# B&R Automation Studio project Panasonic_LinkaPowerCP2_A2021055 (part 32)

#### Main.st - Init, cyclic, exit code
```iecst
PROGRAM _INIT

	//Init parametre serva zdvihu aplikatora//
	P4_Etiketovacka.ServoZdvihuAplikatora.Parameters.Override:= 100;
	P4_Etiketovacka.PAR.ZdvihAplikatora_JoggRychlost:= 5;
	P4_Etiketovacka.ServoZdvihuAplikatora.Command.TorqueLimitation:= TRUE;
	P4_Etiketovacka.ServoZdvihuAplikatora.Parameters.Torque:= 1.0;

END_PROGRAM

PROGRAM _CYCLIC

	//Volanie funkcie SequenceControl//
	SequenceControl(SC:= SC_P4_Etiketovacka);

	//Volanie podprogramov//
	OvlCentrovacky;
	OvlOtacaniaAplikatora;
	IOLinkKomunikacia;
	COM_Tlaciaren;
	VytvorenieEtikety;

	//Enable serva//
	IF Safety.STAV.P4_ZonaBunky_AKTIVNA AND NOT P4_Etiketovacka.ServoZdvihuAplikatora.Command.ErrReset THEN
		P4_Etiketovacka.ServoZdvihuAplikatora.Command.PowerON:= TRUE;
	ELSE
		P4_Etiketovacka.ServoZdvihuAplikatora.Command.PowerON:= FALSE;
	END_IF

	//Zaokrúhlenie aktuálnej pozície serva zdvihu//
	ServoZdvihu_AktualPosition_UDINT:= REAL_TO_UDINT(P4_Etiketovacka.ServoZdvihuAplikatora.Status.ActPosition);

	//Reset poruchy serva//
	IF EDGEPOS(Safety.STAV.P4_ZonaBunky_AKTIVNA)THEN
		P4_Etiketovacka.ServoZdvihuAplikatora.Command.ErrReset:= TRUE;
	END_IF

	CasResetServo_1.IN:= P4_Etiketovacka.ServoZdvihuAplikatora.Command.ErrReset;
	IF CasResetServo_1.Q AND NOT P4_Etiketovacka.ServoZdvihuAplikatora.Status.Error THEN
		P4_Etiketovacka.ServoZdvihuAplikatora.Command.ErrReset:= FALSE;
	END_IF

	CasResetServo_1.PT:= T#500ms;
	CasResetServo_1();

	//Reset sekcie //
	IF P4_Etiketovacka.Reset THEN
		SC_P4_Etiketovacka.Step:= 0;
		P4_Etiketovacka.ServoZdvihuAplikatora.Command.ErrReset:= TRUE;
		P4_Etiketovacka.Reset:= FALSE;
	ELSIF NOT Safety.STAV.Linka_ZonaCS_AKTIVNA AND NOT P4_Etiketovacka.Automat THEN
		SC_P4_Etiketovacka.Step:= 0;
	ELSIF NOT Safety.STAV.Linka_ZonaCS_AKTIVNA AND P4_Etiketovacka.Automat THEN
		P4_Pracovisko.STAV.Porucha_ST5:= TRUE;
	END_IF

	//Ukončenie komunikácie pri poruche//
	IF P4_Pracovisko.STAV.Porucha_ST5 AND NOT Triger_0 THEN
		Triger_0:= TRUE;
		IF P4_Etiketovacka.STAV.VyrobaZacala THEN
			Paletka[i].PAR.StavPowerCP:= 'FAIL';
			Paletka[i].STAV.StavPaletky:= 'NG';
			P4_Etiketovacka.KoniecCyklu:= TRUE;
			SC_P4_Etiketovacka.ResetStep:= TRUE;
			SC_P4_Etiketovacka.Step:= 550;
		ELSE
			SC_P4_Etiketovacka.ResetStep:= TRUE;
			SC_P4_Etiketovacka.Step:= 0;
		END_IF
	END_IF

	IF NOT P4_Pracovisko.STAV.Porucha_ST5 THEN
		Triger_0:= FALSE;
	END_IF

	CASE SC_P4_Etiketovacka.Step OF

		0:
			SC_P4_Etiketovacka.StepName:='0 - Nulovanie';
			SC_OvlCentrovacky.Step:= 0;
			SC_OvlOtacaniaAplikatora.Step:= 0;
			P4_Etiketovacka.Automat:= FALSE;
			P4_Etiketovacka.KoniecCyklu:= FALSE;
			P4_Etiketovacka.Manual:= FALSE;
			P4_Etiketovacka.STAV.PoINIT:= FALSE;
			P4_Etiketovacka.STAV.VyrobaZacala:= FALSE;
			P4_Etiketovacka.STAV.VstupnaKamerovaKontrola:= FALSE;
			P4_Etiketovacka.OUT.ZasunStoper:= FALSE;
			P4_Etiketovacka.OUT.Centrovanie_VYSUN:= FALSE;
			P4_Etiketovacka.OUT.Centrovanie_ZASUN:= TRUE;
			P4_Etiketovacka.OUT.Aplikator_VYSUN:= FALSE;
			P4_Etiketovacka.OUT.Aplikator_OtocVPRED:= FALSE;
			P4_Etiketovacka.OUT.Aplikator_OtocVZAD:= FALSE;
			P4_Etiketovacka.OUT.OfukEtikety_ON:= FALSE;
			P4_Etiketovacka.OUT.PritlakPowerCP_VYSUN:= FALSE;
			P4_Etiketovacka.OUT.PrisavanieEtikety_ON:= FALSE;
			P4_Etiketovacka.OUT.PrisavanieEtikety_OFF:= TRUE;
			P4_Etiketovacka.RFID_hlava.PrecitajChipRFID:= FALSE;

			P4_Etiketovacka.ServoZdvihuAplikatora.Command.JogNeg:= FALSE;
			P4_Etiketovacka.ServoZdvihuAplikatora.Command.JogPos:= FALSE;
			P4_Etiketovacka.ServoZdvihuAplikatora.Command.MoveAdditive:= FALSE;
			P4_Etiketovacka.ServoZdvihuAplikatora.Command.MovePosition:= FALSE;
			IF NOT P4_Etiketovacka.ServoZdvihuAplikatora.Status.StandStill THEN
				P4_Etiketovacka.ServoZdvihuAplikatora.Command.Stop:= TRUE;
			END_IF

			P4_Etiketovacka.CMD.RR_ZdvihAplikatora_DOLE:= FALSE;
			P4_Etiketovacka.CMD.RR_ZdvihAplikatora_HORE:= FALSE;
			P4_Etiketovacka.CMD.RR_NalepEtiketu:= FALSE;
			P4_Etiketovacka.STAV.RR_SekvenciaEtiketovania_BUSY:= FALSE;
			P4_Etiketovacka.CMD.RR_VysunCentrovanie:= FALSE;
			P4_Etiketovacka.CMD.RR_PrisavanieEtikety:= FALSE;

			CAM14.CMD.Triger:= FALSE;
			CAM14.STAV.Results_READY:= FALSE;

			CAM15.CMD.Triger:= FALSE;
			CAM15.STAV.Results_READY:= FALSE;
			FTP_CAM15.CMD.OdosliFotku:= FALSE;
			FTP_CAM15.CMD.VymazFotku:= FALSE;

			TRCB_P4_Etiketovacka_ST9.CMD.VyziadajStavPaletky_TYP1:= FALSE;
			TRCB_P4_Etiketovacka_ST9.CMD.PriradQRkodFiltra_TYP3:= FALSE;
			TRCB_P4_Etiketovacka_ST9.CMD.OdosliStavPaletky_TYP2:= FALSE;
			TRCB_P4_Etiketovacka_ST9.CMD.VyziadajCisloEtikety_TYP0:= FALSE;
			TRCB_P4_Etiketovacka_ST9.CMD.VyziadajStavPanatrace_TYP4:= FALSE;

			P4_Etiketov_KAM_Result_Ignoruj:= FALSE;
			P4_Etiketov_KAM_Result_OK:= FALSE;
			P4_Etiketov_KAM_Result_NG:= FALSE;
			P34_Vizu.ZobrazHL1_ST9:= FALSE;
			P34_Vizu.ZobrazHL2_ST9:= FALSE;
			P34_Vizu.ZobrazHL3_ST9:= FALSE;
			P34_Vizu.ZobrazHL4_ST9:= FALSE;
			TRCB_P4_Etiketov_OpatovnyDopyt:= FALSE;
			TRCB_P4_Etiketov_PaletkaNG:= FALSE;
			PocetTrigrovKamery:= 0;
			PocetDopytovNaServer:= 0;
			CisloFotky:= 0;
			TestovaciKus:= FALSE;
			P4_Etiketovacka.STAV.PowerCP_ZhodaQRkodu_OK:= FALSE;
			P4_Etiketovacka.STAV.Etiketa_ZhodaQRkodu_OK:= FALSE;
			P4_Etiketovacka.STAV.PrebiehaVyvezeniePaletky:= FALSE;
			P4_ZdvizkaZaFunkcTestA.STAV.PrebiehaVyvezeniePaletky:= FALSE;
			P4_Etiketovanie_Taktime.IN.START_MeraniaCasu:= FALSE;
			P4_Etiketovanie_Taktime.IN.START_MeraniaStratovehoCasu:= FALSE;

			Tlaciaren.CMD.VytlacEtiketu:= FALSE;

			IF Safety.STAV.Linka_ZonaCS_AKTIVNA AND
				Safety.STAV.P4_ZonaBunky_AKTIVNA AND
				(P4_Etiketovacka.ServoZdvihuAplikatora.Status.Ready AND P4_Etiketovacka.ServoZdvihuAplikatora.Status.StandStill) AND
				P4_Pracovisko.STAV.HardwareBunky_OK AND
				NOT P4_Pracovisko.STAV.Porucha_ST1 AND
				NOT P4_Pracovisko.STAV.Porucha_ST2 AND
				NOT P4_Pracovisko.STAV.Porucha_ST3 AND
				NOT P4_Pracovisko.STAV.Porucha_ST4 AND
				NOT P4_Pracovisko.STAV.Porucha_ST5 AND
				NOT P4_Pracovisko.STAV.Porucha_ST6 THEN
				P4_Etiketovacka.ServoZdvihuAplikatora.Command.Stop:= FALSE;
				SC_P4_Etiketovacka.ResetStep:= TRUE;
				SC_P4_Etiketovacka.Step:= 1;
			END_IF

		1:
			SC_P4_Etiketovacka.StepName:='1 - Cakam na spustenie vyroby';
			P4_Etiketovacka.KoniecCyklu:= FALSE;
			IF P4_Etiketovacka.Automat THEN
				SC_P4_Etiketovacka.Step:= 2;
			ELSIF P4_Etiketovacka.Manual THEN
				SC_P4_Etiketovacka.Step:= 700;
			END_IF

			//********************************************************Inicializácia****************************************************************************//

		2:
			SC_P4_Etiketovacka.StepName:='2 - Inicializacia - cakam na spustenie inicializacie';
			SC_P4_Etiketovacka.IdleTime.PT:= T#4s;
			SC_P4_Etiketovacka.AlarmTime.PT:= T#5s;

			P4_Etiketovacka.ServoZdvihuAplikatora.Parameters.Acc:= P34_RemPremenne.P4_ZdvihEtiketovacky_Acc;
			P4_Etiketovacka.ServoZdvihuAplikatora.Parameters.Dcc:= P34_RemPremenne.P4_ZdvihEtiketovacky_Dcc;
			P4_Etiketovacka.ServoZdvihuAplikatora.Parameters.Torque:= 1.0;

			IF P4_Dopravniky.STAV.PoINIT THEN
				SC_P4_Etiketovacka.ResetStep:= TRUE;
				SC_P4_Etiketovacka.Step:= 3;
			END_IF

		3:
			SC_P4_Etiketovacka.StepName:='3 - Inicializacia - vymazanie adresara kamery CAM15';
			SC_P4_Etiketovacka.IdleTime.PT:= T#4s;
			SC_P4_Etiketovacka.AlarmTime.PT:= T#5s;

			IF NOT SC_P4_Etiketovacka.Switch1 THEN
				FTP_CAM15.CMD.VymazFotku:= TRUE;
				SC_P4_Etiketovacka.Switch1:= TRUE;
			END_IF

			IF FTP_CAM15.STATUS.KomunikaciaUkoncena THEN
				FTP_CAM15.CMD.VymazFotku:= FALSE;
				SC_P4_Etiketovacka.ResetStep:= TRUE;
				SC_P4_Etiketovacka.Step:= 5;
			ELSIF FTP_CAM15.STATUS.KomunikaciaError THEN
				P34_Alarmy[434]:= TRUE;
				P4_Pracovisko.STAV.Porucha_ST5:= TRUE;
			END_IF

		5:
			SC_P4_Etiketovacka.StepName:='5 - Inicializacia - kontrola otocenia aplikatora';
			SC_P4_Etiketovacka.IdleTime.PT:= T#2s;
			SC_P4_Etiketovacka.AlarmTime.PT:= T#5s;

			IF P4_Etiketovacka.IN.Aplikator_OtocenyVZAD THEN
				SC_P4_Etiketovacka.ResetStep:= TRUE;
				SC_P4_Etiketovacka.Step:= 13;
			ELSE
				SC_P4_Etiketovacka.ResetStep:= TRUE;
				SC_P4_Etiketovacka.Step:= 8;
			END_IF

		8:
			SC_P4_Etiketovacka.StepName:='8 - Inicializacia - zdvih aplikatora do pozicie otocenia aplikatora';
			SC_P4_Etiketovacka.IdleTime.PT:= T#2s;
			SC_P4_Etiketovacka.AlarmTime.PT:= T#5s;

			P4_Etiketovacka.ServoZdvihuAplikatora.Parameters.Velocity:= P34_RemPremenne.P4_Etiketov_RychlZdvihuAplikat/1000;
			P4_Etiketovacka.ServoZdvihuAplikatora.Parameters.Position:= 250;

			IF NOT SC_P4_Etiketovacka.Switch1 THEN
				P4_Etiketovacka.ServoZdvihuAplikatora.Command.MovePosition:= TRUE;
				SC_P4_Etiketovacka.Switch1:= TRUE;
			END_IF

			IF P4_Etiketovacka.ServoZdvihuAplikatora.Status.InPosition THEN
				P4_Etiketovacka.ServoZdvihuAplikatora.Command.MovePosition:= FALSE;
				SC_P4_Etiketovacka.ResetStep:= TRUE;
				SC_P4_Etiketovacka.Step:= 10;
			END_IF

		10:
			SC_P4_Etiketovacka.StepName:='10 - Inicializacia - otocenia aplikatora vzad';
			SC_P4_Etiketovacka.IdleTime.PT:= T#2s;
			SC_P4_Etiketovacka.AlarmTime.PT:= T#5s;

			IF NOT SC_P4_Etiketovacka.Switch1 THEN
				OtocAplikator_VZAD:= TRUE;
				SC_P4_Etiketovacka.Switch1:= TRUE;
			END_IF

			IF P4_Etiketovacka.IN.Aplikator_OtocenyVZAD THEN
				SC_P4_Etiketovacka.ResetStep:= TRUE;
				SC_P4_Etiketovacka.Step:= 13;
			END_IF

		13:
			SC_P4_Etiketovacka.StepName:='13 - Inicializacia - presun zdvihu aplikatora do pozicie odoberania etikety';
			SC_P4_Etiketovacka.IdleTime.PT:= T#2s;
			SC_P4_Etiketovacka.AlarmTime.PT:= T#5s;

			P4_Etiketovacka.ServoZdvihuAplikatora.Parameters.Velocity:= P34_RemPremenne.P4_Etiketov_RychlZdvihuAplikat/1000;
			P4_Etiketovacka.ServoZdvihuAplikatora.Parameters.Position:= P34_RemPremenne.P4_Etiketovacka_PozOdoberEtikety;
			ServoZdvihu_ZadanaPozicia_UDINT:= REAL_TO_UDINT(P34_RemPremenne.P4_Etiketovacka_PozOdoberEtikety);

			IF NOT SC_P4_Etiketovacka.Switch1 THEN
				P4_Etiketovacka.ServoZdvihuAplikatora.Command.MovePosition:= TRUE;
				SC_P4_Etiketovacka.Switch1:= TRUE;
			END_IF

			IF P4_Etiketovacka.ServoZdvihuAplikatora.Status.InPosition AND (ServoZdvihu_AktualPosition_UDINT = ServoZdvihu_ZadanaPozicia_UDINT) THEN
				P4_Etiketovacka.ServoZdvihuAplikatora.Command.MovePosition:= FALSE;
				SC_P4_Etiketovacka.ResetStep:= TRUE;
				SC_P4_Etiketovacka.Step:= 15;
			END_IF

		15:
			SC_P4_Etiketovacka.StepName:='15 - Inicializacia - zasunutie centrovacky';
			SC_P4_Etiketovacka.IdleTime.PT:= T#4s;
			SC_P4_Etiketovacka.AlarmTime.PT:= T#5s;

			IF NOT SC_P4_Etiketovacka.Switch1 THEN
				Centrovacku_ZASUN:= TRUE;
				SC_P4_Etiketovacka.Switch1:= TRUE;
			END_IF

			IF P4_Etiketovacka.IN.Centrovanie_ZASUNUTE THEN
				SC_P4_Etiketovacka.ResetStep:= TRUE;
				SC_P4_Etiketovacka.Step:= 18;
			END_IF

		18:
			SC_P4_Etiketovacka.StepName:='18 - Inicializacia - hladanie paletky';
			SC_P4_Etiketovacka.IdleTime.PT:= T#5s;
			SC_P4_Etiketovacka.AlarmTime.PT:= T#5s;
			SC_P4_Etiketovacka.IdleTime.IN:= TRUE;

			IF P4_Etiketovacka.RFID_hlava.PritomnostPaletky THEN
				SC_P4_Etiketovacka.ResetStep:= TRUE;
				SC_P4_Etiketovacka.Step:= 20;
			ELSIF SC_P4_Etiketovacka.IdleTime.Q THEN
				P4_Etiketovacka.STAV.PoINIT:= TRUE;
				SC_P4_Etiketovacka.ResetStep:= TRUE;
				SC_P4_Etiketovacka.Step:= 100;
			END_IF

		20:
			SC_P4_Etiketovacka.StepName:='20 - Inicializacia - precitanie cisla paletky';
			SC_P4_Etiketovacka.IdleTime.PT:= T#200ms;
			SC_P4_Etiketovacka.AlarmTime.PT:= T#5s;

			SC_P4_Etiketovacka.IdleTime.IN:= P4_Etiketovacka.RFID_hlava.PritomnostPaletky;

			IF SC_P4_Etiketovacka.IdleTime.Q AND NOT SC_P4_Etiketovacka.Switch1 THEN
				P4_Etiketovacka.RFID_hlava.PrecitajChipRFID:= TRUE;
				i:= 0;
				SC_P4_Etiketovacka.Switch1:= TRUE;
			END_IF

			IF P4_Etiketovacka.RFID_hlava.Stav_CitanieZapis_OK AND P4_Etiketovacka.RFID_hlava.PrecitaneCisloPaletky <> 0 THEN
				i:= P4_Etiketovacka.RFID_hlava.PrecitaneCisloPaletky;
				P4_Etiketovacka.PAR.CisloPaletky:= P4_Etiketovacka.RFID_hlava.PrecitaneCisloPaletky;
				P4_Etiketovacka.RFID_hlava.PrecitajChipRFID:= FALSE;
				SC_P4_Etiketovacka.ResetStep:= TRUE;
				SC_P4_Etiketovacka.Step:= 23;
			END_IF

		23:
			SC_P4_Etiketovacka.StepName:='23 - Inicializacia - priradenie indexu paletky na zaklade precitanej hodnoty';
			SC_P4_Etiketovacka.IdleTime.PT:= T#200ms;
			SC_P4_Etiketovacka.AlarmTime.PT:= T#5s;

			IF i<> 0 THEN
				P4_Etiketovacka.PAR.CisloPaletky_STRING:= USINT_TO_STRING(i);
				Paletka[i].PAR.CisloPaletky:= USINT_TO_STRING(i);
				SC_P4_Etiketovacka.ResetStep:= TRUE;
				SC_P4_Etiketovacka.Step:= 30;
			ELSE
				P34_Alarmy[406]:= TRUE;
				P4_Pracovisko.STAV.Porucha_ST5:= TRUE;
			END_IF

		30:
			SC_P4_Etiketovacka.StepName:='30 - Inicializacia - kontrola stavu paletky';
			SC_P4_Etiketovacka.IdleTime.PT:= T#200ms;
			SC_P4_Etiketovacka.AlarmTime.PT:= T#5s;

			IF Paletka[i].STAV.StavPaletky = '' THEN
				Paletka[i].STAV.StavPaletky:= 'NG';
				SC_P4_Etiketovacka.ResetStep:= TRUE;
				SC_P4_Etiketovacka.Step:= 560;
			ELSIF Paletka[i].STAV.StavPaletky = 'PRECH' THEN
				P4_Etiketovacka.STAV.PoINIT:= TRUE;
				SC_P4_Etiketovacka.ResetStep:= TRUE;
				SC_P4_Etiketovacka.Step:= 560;
			ELSIF Paletka[i].STAV.StavPaletky = 'TEST' AND Paletka[i].STAV.CisloTestovacejStanice = 'ST_9' THEN
				TestovaciKus:= TRUE;
			ELSIF Paletka[i].STAV.StavPaletky = 'TEST' AND Paletka[i].STAV.CisloTestovacejStanice <> 'ST_9' THEN
				P4_Etiketovacka.STAV.PoINIT:= TRUE;
				SC_P4_Etiketovacka.ResetStep:= TRUE;
				SC_P4_Etiketovacka.Step:= 560;
			ELSIF Paletka[i].STAV.StavPaletky = 'REV' AND Paletka[i].STAV.CisloRevorkovejStanice = 'ST_9' THEN
				Paletka[i].STAV.StavPaletky:= 'OK';
				SC_P4_Etiketovacka.ResetStep:= TRUE;
				SC_P4_Etiketovacka.Step:= 33;
			ELSIF Paletka[i].STAV.StavPaletky = 'REV' AND Paletka[i].STAV.CisloRevorkovejStanice <> 'ST_9' THEN
				P4_Etiketovacka.STAV.PoINIT:= TRUE;
				SC_P4_Etiketovacka.ResetStep:= TRUE;
				SC_P4_Etiketovacka.Step:= 560;
			ELSIF Paletka[i].STAV.StavPaletky = 'OK' THEN
				SC_P4_Etiketovacka.ResetStep:= TRUE;
				SC_P4_Etiketovacka.Step:= 33;
			ELSIF Paletka[i].STAV.StavPaletky = 'NG' THEN
				P4_Etiketovacka.STAV.PoINIT:= TRUE;
				SC_P4_Etiketovacka.ResetStep:= TRUE;
				SC_P4_Etiketovacka.Step:= 560;
			END_IF

		33:
			SC_P4_Etiketovacka.StepName:='33 - Inicializacia - kontrola uzavretia komunikacie';
			SC_P4_Etiketovacka.IdleTime.PT:= T#200ms;
			SC_P4_Etiketovacka.AlarmTime.PT:= T#5s;

			IF Paletka[i].STAV.Komunikacia_DONE THEN
				P4_Etiketovacka.STAV.PoINIT:= TRUE;
				SC_P4_Etiketovacka.ResetStep:= TRUE;
				SC_P4_Etiketovacka.Step:= 560;
			ELSE
				P4_Etiketovacka.STAV.PoINIT:= TRUE;
				P4_Etiketovacka.STAV.VstupnaKamerovaKontrola:= TRUE;
				SC_P4_Etiketovacka.ResetStep:= TRUE;
				SC_P4_Etiketovacka.Step:= 100;
			END_IF

			//********************************************************Automatický režim****************************************************************************//

		100:
			SC_P4_Etiketovacka.StepName:='100 - Automaticky Rezim - cakam na príchod paletky na stoper';
			SC_P4_Etiketovacka.IdleTime.PT:= T#200ms;
			SC_P4_Etiketovacka.AlarmTime.PT:= T#5s;

			SC_P4_Etiketovacka.IdleTime.IN:= P4_Etiketovacka.RFID_hlava.PritomnostPaletky;

			P4_Etiketovacka.ServoZdvihuAplikatora.Parameters.Acc:= P34_RemPremenne.P4_ZdvihEtiketovacky_Acc;
			P4_Etiketovacka.ServoZdvihuAplikatora.Parameters.Dcc:= P34_RemPremenne.P4_ZdvihEtiketovacky_Dcc;
			P4_Etiketovacka.ServoZdvihuAplikatora.Parameters.Torque:= 1.0;

			IF P4_Etiketovacka.RFID_hlava.PritomnostPaletky THEN
				P4_ZdvizkaZaFunkcTestA.STAV.PrebiehaVyvezeniePaletky:= FALSE;
			END_IF

			IF NOT SC_P4_Etiketovacka.Switch1 AND P4_Etiketovacka.RFID_hlava.PritomnostPaletky THEN
				P4_Etiketovanie_Taktime.IN.START_MeraniaCasu:= TRUE;
				P4_Etiketovanie_Taktime.IN.ZAPIS_MeraniaCasu:= TRUE;
				P4_Etiketovanie_Taktime.IN.ZAPIS_StratovyCas:= TRUE;
				Buffer_13.Hodnota:= P4_Etiketovanie_Taktime.OUT.StratoveSekundy;
				Buffer_13.ZapisHodnotu:= TRUE;
				SC_P4_Etiketovacka.Switch1:= TRUE;
			END_IF

			IF P4_Etiketovacka.KoniecCyklu AND NOT P4_ZdvizkaZaFunkcTestA.Automat THEN
				SC_P4_Etiketovacka.ResetStep:= TRUE;
				SC_P4_Etiketovacka.Step:= 0;
			ELSIF SC_P4_Etiketovacka.IdleTime.Q THEN
				SC_P4_Etiketovacka.ResetStep:= TRUE;
				SC_P4_Etiketovacka.Step:= 101;
			END_IF

		101:
			SC_P4_Etiketovacka.StepName:='101 - Automaticky Rezim - precitanie cisla paletky';
			SC_P4_Etiketovacka.IdleTime.PT:= T#500ms;
			SC_P4_Etiketovacka.AlarmTime.PT:= T#5s;
			SC_P4_Etiketovacka.IdleTime.IN:= TRUE;

			IF NOT SC_P4_Etiketovacka.Switch1 THEN
				i:= 0;
				P4_Etiketovacka.RFID_hlava.PrecitajChipRFID:= TRUE;
				SC_P4_Etiketovacka.Switch1:= TRUE;
			END_IF

			IF P4_Etiketovacka.RFID_hlava.Stav_CitanieZapis_OK AND P4_Etiketovacka.RFID_hlava.PrecitaneCisloPaletky <> 0 THEN
				i:= P4_Etiketovacka.RFID_hlava.PrecitaneCisloPaletky;
				P4_Etiketovacka.PAR.CisloPaletky:= P4_Etiketovacka.RFID_hlava.PrecitaneCisloPaletky;
				P4_Etiketovacka.RFID_hlava.PrecitajChipRFID:= FALSE;
				SC_P4_Etiketovacka.ResetStep:= TRUE;
				SC_P4_Etiketovacka.Step:= 102;
			END_IF

		102:
			SC_P4_Etiketovacka.StepName:='102 - Automaticky Rezim - priradenie indexu paletky na zaklade precitanej hodnoty';
			SC_P4_Etiketovacka.IdleTime.PT:= T#200ms;
			SC_P4_Etiketovacka.AlarmTime.PT:= T#5s;

			IF i<> 0 THEN
				P4_Etiketovacka.PAR.CisloPaletky_STRING:= USINT_TO_STRING(i);
				Paletka[i].PAR.CisloPaletky:= USINT_TO_STRING(i);
				SC_P4_Etiketovacka.ResetStep:= TRUE;
				SC_P4_Etiketovacka.Step:= 103;
			ELSE
				P34_Alarmy[406]:= TRUE;
				P4_Pracovisko.STAV.Porucha_ST5:= TRUE;
			END_IF

		103:
			SC_P4_Etiketovacka.StepName:='103 - Automaticky Rezim - kontrola stavu paletky';
			SC_P4_Etiketovacka.IdleTime.PT:= T#200ms;
			SC_P4_Etiketovacka.AlarmTime.PT:= T#5s;

			IF Paletka[i].STAV.StavPaletky = '' THEN
				Paletka[i].STAV.StavPaletky:= 'NG';
				SC_P4_Etiketovacka.ResetStep:= TRUE;
				SC_P4_Etiketovacka.Step:= 560;
			ELSIF Paletka[i].STAV.StavPaletky = 'PRECH' THEN
				SC_P4_Etiketovacka.ResetStep:= TRUE;
				SC_P4_Etiketovacka.Step:= 560;
			ELSIF Paletka[i].STAV.StavPaletky = 'TEST' AND Paletka[i].STAV.CisloTestovacejStanice = 'ST_9' THEN
				TestovaciKus:= TRUE;
			ELSIF Paletka[i].STAV.StavPaletky = 'TEST' AND Paletka[i].STAV.CisloTestovacejStanice <> 'ST_9' THEN
				SC_P4_Etiketovacka.ResetStep:= TRUE;
				SC_P4_Etiketovacka.Step:= 560;
			ELSIF Paletka[i].STAV.StavPaletky = 'REV' AND Paletka[i].STAV.CisloRevorkovejStanice = 'ST_9' THEN
				Paletka[i].STAV.StavPaletky:= 'OK';
				SC_P4_Etiketovacka.ResetStep:= TRUE;
				SC_P4_Etiketovacka.Step:= 105;
			ELSIF Paletka[i].STAV.StavPaletky = 'REV' AND Paletka[i].STAV.CisloRevorkovejStanice <> 'ST_9' THEN
				SC_P4_Etiketovacka.ResetStep:= TRUE;
				SC_P4_Etiketovacka.Step:= 560;
			ELSIF Paletka[i].STAV.StavPaletky = 'OK' THEN
				SC_P4_Etiketovacka.ResetStep:= TRUE;
				SC_P4_Etiketovacka.Step:= 105;
			ELSIF Paletka[i].STAV.StavPaletky = 'NG' THEN
				SC_P4_Etiketovacka.ResetStep:= TRUE;
				SC_P4_Etiketovacka.Step:= 560;
			END_IF

		105:
			SC_P4_Etiketovacka.StepName:='105 - Automaticky Rezim - vyziadanie stavu komunikacie zo serverom';
			SC_P4_Etiketovacka.IdleTime.PT:= T#200ms;
			SC_P4_Etiketovacka.AlarmTime.PT:= T#10s;

			IF Linka.KOM_Panatrace_OFF THEN
				SC_P4_Etiketovacka.ResetStep:= TRUE;
				SC_P4_Etiketovacka.Step:= 118;
			ELSIF NOT SC_P4_Etiketovacka.Switch1 AND TRCB_P4_Etiketovacka_ST9.STATUS.KOM_READY THEN
				TRCB_P4_Etiketovacka_ST9.CMD.VyziadajStavPanatrace_TYP4:= TRUE;
				Centrovacku_VYSUN:= TRUE;
				(*P4_Etiketovanie_Taktime.IN.START_MeraniaStratovehoCasu:= TRUE;*)
				SC_P4_Etiketovacka.Switch1:= TRUE;
			END_IF

			IF TRCB_P4_Etiketovacka_ST9.STATUS.KomunikaciaUkoncena THEN
				TRCB_P4_Etiketovacka_ST9.CMD.VyziadajStavPanatrace_TYP4:= FALSE;
				P4_Etiketovanie_Taktime.IN.START_MeraniaStratovehoCasu:= FALSE;
				SC_P4_Etiketovacka.ResetStep:= TRUE;
				SC_P4_Etiketovacka.Step:= 106;
			ELSIF TRCB_P4_Etiketovacka_ST9.STATUS.KomunikaciaError THEN
				TRCB_P4_Etiketovacka_ST9.CMD.VyziadajStavPanatrace_TYP4:= FALSE;
				P4_Etiketovanie_Taktime.IN.START_MeraniaStratovehoCasu:= FALSE;
				SC_P4_Etiketovacka.ResetStep:= TRUE;
				SC_P4_Etiketovacka.Step:= 107;
			END_IF

		106:
			SC_P4_Etiketovacka.StepName:='106 - Automaticky Rezim - kontrola odpovede servera';
			SC_P4_Etiketovacka.IdleTime.PT:= T#200ms;
			SC_P4_Etiketovacka.AlarmTime.PT:= T#5s;

			IF NOT TRCB_P4_Etiketovacka_ST9.STATUS.KomunikaciaUkoncena THEN
				IF TRCB_P4_Etiketovacka_ST9.OUTPUTS.DruhCinnostiNaPaletke = '0;Generating' THEN
					SC_P4_Etiketovacka.ResetStep:= TRUE;
					SC_P4_Etiketovacka.Step:= 107;
				ELSIF TRCB_P4_Etiketovacka_ST9.OUTPUTS.DruhCinnostiNaPaletke = '1;Request' THEN
					SC_P4_Etiketovacka.ResetStep:= TRUE;
					SC_P4_Etiketovacka.Step:= 108;
				ELSIF TRCB_P4_Etiketovacka_ST9.OUTPUTS.DruhCinnostiNaPaletke = '2;Report' THEN
					SC_P4_Etiketovacka.ResetStep:= TRUE;
					SC_P4_Etiketovacka.Step:= 118;
				ELSIF TRCB_P4_Etiketovacka_ST9.OUTPUTS.DruhCinnostiNaPaletke = '3;Wedding' THEN
					SC_P4_Etiketovacka.ResetStep:= TRUE;
					SC_P4_Etiketovacka.Step:= 107;
				ELSIF TRCB_P4_Etiketovacka_ST9.OUTPUTS.DruhCinnostiNaPaletke = '4;Status' THEN
					SC_P4_Etiketovacka.ResetStep:= TRUE;
					SC_P4_Etiketovacka.Step:= 107;
				ELSIF TRCB_P4_Etiketovacka_ST9.OUTPUTS.DruhCinnostiNaPaletke = '5;' THEN
					SC_P4_Etiketovacka.ResetStep:= TRUE;
					SC_P4_Etiketovacka.Step:= 107;
				ELSE
					SC_P4_Etiketovacka.ResetStep:= TRUE;
					SC_P4_Etiketovacka.Step:= 107;
				END_IF
			END_IF

		107:
			SC_P4_Etiketovacka.StepName:='107 - Automaticky Rezim - rozhodnutie obsluhy po chybe komunikacie s Panatrace';
			SC_P4_Etiketovacka.IdleTime.PT:= T#200ms;
			SC_P4_Etiketovacka.AlarmTime.PT:= T#5s;

			P34_Vizu.ZobrazHL4_ST9:= TRUE;

			IF TRCB_P4_Etiketov_OpatovnyDopyt THEN
				TRCB_P4_Etiketov_OpatovnyDopyt:= FALSE;
				P34_Vizu.ZobrazHL4_ST9:= FALSE;
				SC_P4_Etiketovacka.ResetStep:= TRUE;
				SC_P4_Etiketovacka.Step:= 105;
			ELSIF TRCB_P4_Etiketov_PaletkaNG THEN
				TRCB_P4_Etiketov_PaletkaNG:= FALSE;
				P34_Vizu.ZobrazHL4_ST9:= FALSE;
				Paletka[i].STAV.StavPaletky := 'NG';
				SC_P4_Etiketovacka.ResetStep:= TRUE;
				SC_P4_Etiketovacka.Step:= 116;
			END_IF

		108:
			SC_P4_Etiketovacka.StepName:='108 - Automaticky Rezim - vyziadanie stavu paletky zo servera, zacentrovanie paletky';
			SC_P4_Etiketovacka.IdleTime.PT:= T#200ms;
			SC_P4_Etiketovacka.AlarmTime.PT:= T#10s;
			SC_P4_Etiketovacka.IdleTime.IN:= TRUE;

			IF NOT SC_P4_Etiketovacka.Switch1 AND TRCB_P4_Etiketovacka_ST9.STATUS.KOM_READY THEN
				TRCB_P4_Etiketovacka_ST9.CMD.VyziadajStavPaletky_TYP1:= TRUE;
				(*P4_Etiketovanie_Taktime.IN.START_MeraniaStratovehoCasu:= TRUE;*)
				SC_P4_Etiketovacka.Switch1:= TRUE;
			END_IF

			IF TRCB_P4_Etiketovacka_ST9.STATUS.KomunikaciaUkoncena THEN
				TRCB_P4_Etiketovacka_ST9.CMD.VyziadajStavPaletky_TYP1:= FALSE;
				P4_Etiketovanie_Taktime.IN.START_MeraniaStratovehoCasu:= FALSE;
				SC_P4_Etiketovacka.ResetStep:= TRUE;
				SC_P4_Etiketovacka.Step:= 110;
			ELSIF TRCB_P4_Etiketovacka_ST9.STATUS.KomunikaciaError THEN
				TRCB_P4_Etiketovacka_ST9.CMD.VyziadajStavPaletky_TYP1:= FALSE;
				P4_Etiketovanie_Taktime.IN.START_MeraniaStratovehoCasu:= FALSE;
				SC_P4_Etiketovacka.ResetStep:= TRUE;
				SC_P4_Etiketovacka.Step:= 107;
			END_IF

		110:
			SC_P4_Etiketovacka.StepName:='110 - Automaticky Rezim - kontrola odpovede servera';
			SC_P4_Etiketovacka.IdleTime.PT:= T#200ms;
			SC_P4_Etiketovacka.AlarmTime.PT:= T#5s;

			IF NOT TRCB_P4_Etiketovacka_ST9.STATUS.KomunikaciaUkoncena AND P4_Etiketovacka.IN.Centrovanie_VYSUNUTE THEN
				IF TRCB_P4_Etiketovacka_ST9.OUTPUTS.PovolenieCinnostiNaPaletke = 'OK' THEN
					IF TRCB_P4_Etiketovacka_ST9.OUTPUTS.DruhCinnostiNaPaletke = 'PRD;ST9' THEN
						P4_Etiketovacka.OUT.OfukEtikety_ON:= TRUE;
						P4_Etiketovacka.OUT.PrisavanieEtikety_OFF:= FALSE;
						P4_Etiketovacka.OUT.PrisavanieEtikety_ON:= TRUE;
						SC_P4_Etiketovacka.ResetStep:= TRUE;
						SC_P4_Etiketovacka.Step:= 118;
					ELSE
						Paletka[i].STAV.StavPaletky := 'NG';
						SC_P4_Etiketovacka.ResetStep:= TRUE;
						SC_P4_Etiketovacka.Step:= 116;
					END_IF
				ELSIF TRCB_P4_Etiketovacka_ST9.OUTPUTS.PovolenieCinnostiNaPaletke = 'NG' THEN
					SC_P4_Etiketovacka.ResetStep:= TRUE;
					SC_P4_Etiketovacka.Step:= 115;
				END_IF
			END_IF

		115:
			SC_P4_Etiketovacka.StepName:='115 - Automaticky Rezim - rozhodnutie obsluhy po odpovedi panatrace NG';
			SC_P4_Etiketovacka.IdleTime.PT:= T#200ms;
			SC_P4_Etiketovacka.AlarmTime.PT:= T#5s;

			P34_Vizu.ZobrazHL3_ST9:= TRUE;

			IF TRCB_P4_Etiketov_OpatovnyDopyt THEN
				TRCB_P4_Etiketov_OpatovnyDopyt:= FALSE;
				P34_Vizu.ZobrazHL3_ST9:= FALSE;
				SC_P4_Etiketovacka.ResetStep:= TRUE;
				SC_P4_Etiketovacka.Step:= 105;
			ELSIF TRCB_P4_Etiketov_PaletkaNG THEN
				TRCB_P4_Etiketov_PaletkaNG:= FALSE;
				P34_Vizu.ZobrazHL3_ST9:= FALSE;
				Paletka[i].STAV.StavPaletky := 'NG';
				SC_P4_Etiketovacka.ResetStep:= TRUE;
				SC_P4_Etiketovacka.Step:= 116;
			END_IF

		116:
			SC_P4_Etiketovacka.StepName:='116 - Automaticky Rezim - odcentrovanie paletky po odpovedi servera NG';
			SC_P4_Etiketovacka.IdleTime.PT:= T#200ms;
			SC_P4_Etiketovacka.AlarmTime.PT:= T#5s;

			IF NOT SC_P4_Etiketovacka.Switch1 THEN
				Centrovacku_ZASUN:= TRUE;
				SC_P4_Etiketovacka.Switch1:= TRUE;
			END_IF

			IF P4_Etiketovacka.IN.Centrovanie_ZASUNUTE THEN
				SC_P4_Etiketovacka.ResetStep:= TRUE;
				SC_P4_Etiketovacka.Step:= 560;
			END_IF

			//Štart aplikovania etikety//

		118:
			SC_P4_Etiketovacka.StepName:='118 - Automaticky Rezim - zacentrovanie paletky ';
			SC_P4_Etiketovacka.IdleTime.PT:= T#200ms;
			SC_P4_Etiketovacka.AlarmTime.PT:= T#5s;

			IF NOT SC_P4_Etiketovacka.Switch1 THEN
				Centrovacku_VYSUN:= TRUE;
				SC_P4_Etiketovacka.Switch1:= TRUE;
			END_IF

			IF P4_Etiketovacka.IN.Centrovanie_VYSUNUTE THEN
				P4_Etiketovacka.OUT.PritlakPowerCP_VYSUN:= TRUE;
				CAM14.STAV.OldRunCounter:= CAM14.STAV.RunCounter;
				CAM14.STAV.Results_READY:= FALSE;
				IF P4_Etiketovacka.STAV.RR_SekvenciaEtiketovania_BUSY THEN
					SC_P4_Etiketovacka.ResetStep:= TRUE;
					SC_P4_Etiketovacka.Step:= 124;
				ELSE
					SC_P4_Etiketovacka.ResetStep:= TRUE;
					SC_P4_Etiketovacka.Step:= 120;
				END_IF
			END_IF

		120:
			SC_P4_Etiketovacka.StepName:='120 - Automaticky Rezim - precitanie QR kodu na Power CP CAM14';//CAM 14//
			SC_P4_Etiketovacka.IdleTime.PT:= T#5s;
			SC_P4_Etiketovacka.AlarmTime.PT:= T#5s;

			IF NOT SC_P4_Etiketovacka.Switch1 THEN
				CAM14.CMD.Triger:= TRUE;
				P4_Etiketovacka.STAV.PowerCP_ZhodaQRkodu_OK:= FALSE;
				CAM14.RESULT.PowerCP.PrecitanyQRkod_PowerCP:= '';
				SC_P4_Etiketovacka.IdleTime.IN:= TRUE;
				SC_P4_Etiketovacka.Switch1:= TRUE;
			END_IF

			IF CAM14.STAV.Results_READY AND CAM14.STAV.OldRunCounter <> CAM14.STAV.RunCounter THEN
				PocetTrigrovKamery:= 0;
				CAM14.STAV.Results_READY:= FALSE;
				CAM14.STAV.OldRunCounter:= CAM14.STAV.RunCounter;
				SC_P4_Etiketovacka.ResetStep:= TRUE;
				SC_P4_Etiketovacka.Step:= 122;
			ELSIF SC_P4_Etiketovacka.IdleTime.Q AND PocetTrigrovKamery < 5 THEN
				PocetTrigrovKamery:= PocetTrigrovKamery + 1;
				CAM14.CMD.Triger:= FALSE;
				CAM14.STAV.Results_READY:= FALSE;
				CAM14.STAV.OldRunCounter:= CAM14.STAV.RunCounter;
				SC_P4_Etiketovacka.ResetStep:= TRUE;
				SC_P4_Etiketovacka.Step:= 121;
			ELSIF SC_P4_Etiketovacka.IdleTime.Q AND PocetTrigrovKamery >= 5 THEN
				P34_Alarmy[453]:= TRUE;
				P4_Pracovisko.STAV.Porucha_ST5:= TRUE;
			END_IF

		121:
			SC_P4_Etiketovacka.StepName:='121 - Automaticky Rezim - cakam na opatovny triger kamery CAM14';
			SC_P4_Etiketovacka.IdleTime.PT:= T#1s;
			SC_P4_Etiketovacka.AlarmTime.PT:= T#5s;

			SC_P4_Etiketovacka.IdleTime.IN:= TRUE;

			IF SC_P4_Etiketovacka.IdleTime.Q THEN
				SC_P4_Etiketovacka.ResetStep:= TRUE;
				SC_P4_Etiketovacka.Step:= 120;
			END_IF

		122:
			SC_P4_Etiketovacka.StepName:='122 - Automaticky Rezim - kontrola vysledku kamery';
			SC_P4_Etiketovacka.IdleTime.PT:= T#300ms;
			SC_P4_Etiketovacka.AlarmTime.PT:= T#5s;
			SC_P4_Etiketovacka.IdleTime.IN:= TRUE;

			IF Linka.P4_Kamery_OFF THEN
				CAM14.CMD.Triger:= FALSE;
				CAM14.PAR.ResultFotky:= 'PASS';
				SC_P4_Etiketovacka.ResetStep:= TRUE;
				SC_P4_Etiketovacka.Step:= 123;
			ELSIF NOT CAM14.STAV.BUSY AND SC_P4_Etiketovacka.IdleTime.Q THEN
				CAM14.CMD.Triger:= FALSE;
				IF CAM14.RESULT.PowerCP.CitanieQRkodu_PowerCP_OK THEN
					IF Paletka[i].PAR.QRkodPowerCP = CAM14.RESULT.PowerCP.PrecitanyQRkod_PowerCP THEN
						P4_Etiketovacka.STAV.PowerCP_ZhodaQRkodu_OK:= TRUE;
						CAM14.PAR.ResultFotky:= 'PASS';
						SC_P4_Etiketovacka.ResetStep:= TRUE;
						SC_P4_Etiketovacka.Step:= 123;
					ELSE
						CAM14.PAR.ResultFotky:= 'FAIL';
						P4_Etiketovacka.STAV.PowerCP_ZhodaQRkodu_OK:= FALSE;
						SC_P4_Etiketovacka.ResetStep:= TRUE;
						SC_P4_Etiketovacka.Step:= 123;
					END_IF
				ELSE
					CAM14.PAR.ResultFotky:= 'FAIL';
					P4_Etiketovacka.STAV.PowerCP_ZhodaQRkodu_OK:= FALSE;
					SC_P4_Etiketovacka.ResetStep:= TRUE;
					SC_P4_Etiketovacka.Step:= 123;
				END_IF
			END_IF

		123:
			SC_P4_Etiketovacka.StepName:='123 - Automaticky Rezim - rozhodnutie podla kamerovej kontroly paletky';
			SC_P4_Etiketovacka.IdleTime.PT:= T#200ms;
			SC_P4_Etiketovacka.AlarmTime.PT:= T#5s;

			IF CAM14.PAR.ResultFotky = 'PASS' THEN
				SC_P4_Etiketovacka.ResetStep:= TRUE;
				SC_P4_Etiketovacka.Step:= 124;
			ELSIF CAM14.PAR.ResultFotky = 'FAIL' THEN
				P34_Vizu.ZobrazHL1_ST9:= TRUE;
				IF P4_Etiketov_KAM_Result_OK THEN
					P4_Etiketov_KAM_Result_OK:= FALSE;
					CAM14.PAR.ResultFotky:= 'PASS';
					P34_Vizu.ZobrazHL1_ST9:= FALSE;
					SC_P4_Etiketovacka.ResetStep:= TRUE;
					SC_P4_Etiketovacka.Step:= 124;
				ELSIF P4_Etiketov_KAM_Result_NG THEN
					P4_Etiketov_KAM_Result_NG:= FALSE;
					P34_Vizu.ZobrazHL1_ST9:= FALSE;
					Paletka[i].PAR.StavPowerCP:= 'FAIL';
					Paletka[i].STAV.StavPaletky:= 'NG';
					P4_Etiketovacka.OUT.OfukEtikety_ON:= FALSE;
					P4_Etiketovacka.OUT.PrisavanieEtikety_OFF:= TRUE;
					P4_Etiketovacka.OUT.PrisavanieEtikety_ON:= FALSE;
					SC_P4_Etiketovacka.ResetStep:= TRUE;
					SC_P4_Etiketovacka.Step:= 540;
				END_IF
			END_IF

		124:
			SC_P4_Etiketovacka.StepName:='123 - Automaticky Rezim - zapnutie prisavania etikety a spodneho ofuku etikety';
			SC_P4_Etiketovacka.IdleTime.PT:= T#200ms;
			SC_P4_Etiketovacka.AlarmTime.PT:= T#5s;

			P4_Etiketovacka.OUT.OfukEtikety_ON:= TRUE;
			P4_Etiketovacka.OUT.PrisavanieEtikety_OFF:= FALSE;
			P4_Etiketovacka.OUT.PrisavanieEtikety_ON:= TRUE;
			IF P4_Etiketovacka.STAV.RR_SekvenciaEtiketovania_BUSY THEN
				SC_P4_Etiketovacka.ResetStep:= TRUE;
				SC_P4_Etiketovacka.Step:= 138;
			ELSIF Linka.KOM_Panatrace_OFF THEN
				SC_P4_Etiketovacka.ResetStep:= TRUE;
				SC_P4_Etiketovacka.Step:= 138;
			ELSE
				SC_P4_Etiketovacka.ResetStep:= TRUE;
				SC_P4_Etiketovacka.Step:= 127;
			END_IF

		127:
			SC_P4_Etiketovacka.StepName:='127 - Automaticky Rezim - vyziadanie stavu komunikacie zo serverom';
			SC_P4_Etiketovacka.IdleTime.PT:= T#200ms;
			SC_P4_Etiketovacka.AlarmTime.PT:= T#10s;

			IF Linka.KOM_Panatrace_OFF THEN
				SC_P4_Etiketovacka.ResetStep:= TRUE;
				SC_P4_Etiketovacka.Step:= 138;
			ELSIF NOT SC_P4_Etiketovacka.Switch1 THEN
				TRCB_P4_Etiketovacka_ST9.CMD.VyziadajStavPanatrace_TYP4:= TRUE;
				SC_P4_Etiketovacka.Switch1:= TRUE;
			END_IF

			IF TRCB_P4_Etiketovacka_ST9.STATUS.KomunikaciaUkoncena THEN
				TRCB_P4_Etiketovacka_ST9.CMD.VyziadajStavPanatrace_TYP4:= FALSE;
				SC_P4_Etiketovacka.ResetStep:= TRUE;
				SC_P4_Etiketovacka.Step:= 128;
			ELSIF TRCB_P4_Etiketovacka_ST9.STATUS.KomunikaciaError THEN
				TRCB_P4_Etiketovacka_ST9.CMD.VyziadajStavPanatrace_TYP4:= FALSE;
				P34_Alarmy[409]:= TRUE;
				P4_Pracovisko.STAV.Porucha_ST5:= TRUE;
			END_IF

		128:
			SC_P4_Etiketovacka.StepName:='128 - Automaticky Rezim - kontrola odpovede servera';
			SC_P4_Etiketovacka.IdleTime.PT:= T#200ms;
			SC_P4_Etiketovacka.AlarmTime.PT:= T#5s;

			IF NOT TRCB_P4_Etiketovacka_ST9.STATUS.KomunikaciaUkoncena THEN
				IF TRCB_P4_Etiketovacka_ST9.OUTPUTS.DruhCinnostiNaPaletke = '0;Generating' THEN
					SC_P4_Etiketovacka.ResetStep:= TRUE;
					SC_P4_Etiketovacka.Step:= 130;
				ELSIF TRCB_P4_Etiketovacka_ST9.OUTPUTS.DruhCinnostiNaPaletke = '1;Request' THEN
					SC_P4_Etiketovacka.ResetStep:= TRUE;
					SC_P4_Etiketovacka.Step:= 100;
				ELSIF TRCB_P4_Etiketovacka_ST9.OUTPUTS.DruhCinnostiNaPaletke = '2;Report' THEN
					SC_P4_Etiketovacka.ResetStep:= TRUE;
					SC_P4_Etiketovacka.Step:= 130;
				ELSIF TRCB_P4_Etiketovacka_ST9.OUTPUTS.DruhCinnostiNaPaletke = '3;Wedding' THEN
					SC_P4_Etiketovacka.ResetStep:= TRUE;
					SC_P4_Etiketovacka.Step:= 129;
				ELSIF TRCB_P4_Etiketovacka_ST9.OUTPUTS.DruhCinnostiNaPaletke = '4;Status' THEN
					SC_P4_Etiketovacka.ResetStep:= TRUE;
					SC_P4_Etiketovacka.Step:= 129;
				ELSIF TRCB_P4_Etiketovacka_ST9.OUTPUTS.DruhCinnostiNaPaletke = '5;' THEN
					SC_P4_Etiketovacka.ResetStep:= TRUE;
					SC_P4_Etiketovacka.Step:= 129;
				ELSE
					SC_P4_Etiketovacka.ResetStep:= TRUE;
					SC_P4_Etiketovacka.Step:= 129;
				END_IF
			END_IF

		129:
			SC_P4_Etiketovacka.StepName:='129 - Automaticky Rezim - rozhodnutie obsluhy po chybe komunikacie s Panatrace';
			SC_P4_Etiketovacka.IdleTime.PT:= T#200ms;
			SC_P4_Etiketovacka.AlarmTime.PT:= T#5s;

			P34_Vizu.ZobrazHL4_ST9:= TRUE;

			IF TRCB_P4_Etiketov_OpatovnyDopyt THEN
				TRCB_P4_Etiketov_OpatovnyDopyt:= FALSE;
				P34_Vizu.ZobrazHL4_ST9:= FALSE;
				SC_P4_Etiketovacka.ResetStep:= TRUE;
				SC_P4_Etiketovacka.Step:= 127;
			ELSIF TRCB_P4_Etiketov_PaletkaNG THEN
				TRCB_P4_Etiketov_PaletkaNG:= FALSE;
				P34_Vizu.ZobrazHL4_ST9:= FALSE;
				Paletka[i].STAV.StavPaletky := 'NG';
				P4_Etiketovacka.STAV.VyrobaZacala:= FALSE;
				SC_P4_Etiketovacka.ResetStep:= TRUE;
				SC_P4_Etiketovacka.Step:= 560;
			END_IF

		130:
			SC_P4_Etiketovacka.StepName:='130 - Automaticky Rezim - vyziadanie serioveho cisla etikety zo servera';
			SC_P4_Etiketovacka.IdleTime.PT:= T#200ms;
			SC_P4_Etiketovacka.AlarmTime.PT:= T#10s;

			IF NOT SC_P4_Etiketovacka.Switch1 AND TRCB_P4_Etiketovacka_ST9.STATUS.KOM_READY THEN
				SerioveCisloEtikety:= '';
				TRCB_P4_Etiketovacka_ST9.CMD.VyziadajCisloEtikety_TYP0:= TRUE;
				SC_P4_Etiketovacka.Switch1:= TRUE;
			END_IF

			IF TRCB_P4_Etiketovacka_ST9.STATUS.KomunikaciaUkoncena THEN
				TRCB_P4_Etiketovacka_ST9.CMD.VyziadajCisloEtikety_TYP0:= FALSE;
				SC_P4_Etiketovacka.ResetStep:= TRUE;
				SC_P4_Etiketovacka.Step:= 133;
			ELSIF TRCB_P4_Etiketovacka_ST9.STATUS.KomunikaciaError THEN
				TRCB_P4_Etiketovacka_ST9.CMD.VyziadajCisloEtikety_TYP0:= FALSE;
				P34_Alarmy[409]:= TRUE;
				P4_Pracovisko.STAV.Porucha_ST5:= TRUE;
			END_IF

		133:
			SC_P4_Etiketovacka.StepName:='133 - Automaticky Rezim - kontrola odpovede servera';
			SC_P4_Etiketovacka.IdleTime.PT:= T#200ms;
			SC_P4_Etiketovacka.AlarmTime.PT:= T#5s;

			IF NOT TRCB_P4_Etiketovacka_ST9.STATUS.KomunikaciaUkoncena THEN
				Paletka[i].STAV.CisloEtiketyVyziadane:= TRUE;
				IF TRCB_P4_Etiketovacka_ST9.OUTPUTS.PovolenieCinnostiNaPaletke = 'OK' THEN
					SerioveCisloEtikety:= TRCB_P4_Etiketovacka_ST9.OUTPUTS.CisloEtikety;
					SC_P4_Etiketovacka.ResetStep:= TRUE;
					SC_P4_Etiketovacka.Step:= 140;
				ELSIF TRCB_P4_Etiketovacka_ST9.OUTPUTS.PovolenieCinnostiNaPaletke = 'NG' THEN
					Paletka[i].STAV.StavPaletky := 'NG';
					P4_Etiketovacka.OUT.PrisavanieEtikety_ON:= FALSE;
					P4_Etiketovacka.OUT.PrisavanieEtikety_OFF:= TRUE;
					P4_Etiketovacka.OUT.OfukEtikety_ON:= FALSE;
					SC_P4_Etiketovacka.ResetStep:= TRUE;
					SC_P4_Etiketovacka.Step:= 560;
				END_IF
			END_IF

		138:
			SC_P4_Etiketovacka.StepName:='138 - Automaticky Rezim - vytlacenie etikety z PLC';
			SC_P4_Etiketovacka.IdleTime.PT:= T#500ms;
			SC_P4_Etiketovacka.AlarmTime.PT:= T#5s;

			P4_Etiketovacka.OUT.PrisavanieEtikety_ON:= TRUE;
			P4_Etiketovacka.OUT.PrisavanieEtikety_OFF:= FALSE;
			P4_Etiketovacka.OUT.OfukEtikety_ON:= TRUE;
			SC_P4_Etiketovacka.IdleTime.IN:= TRUE;

			IF NOT SC_P4_Etiketovacka.Switch1 AND SC_P4_Etiketovacka.IdleTime.Q THEN
				Tlaciaren.CMD.VytlacEtiketu:= TRUE;
				SC_P4_Etiketovacka.Switch1:= TRUE;
			END_IF

			IF Tlaciaren.STAV.VytlacenieEtikety_OK THEN
				Tlaciaren.CMD.VytlacEtiketu:= FALSE;
				SC_P4_Etiketovacka.ResetStep:= TRUE;
				SC_P4_Etiketovacka.Step:= 140;
			ELSIF Tlaciaren.STAV.VytlacenieEtikety_ERROR THEN
				Tlaciaren.CMD.VytlacEtiketu:= FALSE;
				P34_Alarmy[431]:= TRUE;
				P4_Pracovisko.STAV.Porucha_ST5:= TRUE;
			END_IF

		140:
			SC_P4_Etiketovacka.StepName:='140 - Automaticky Rezim - cakam na vysunutie etikety z tlaciarne, vypnutie ofuku etikety';
			SC_P4_Etiketovacka.IdleTime.PT:= T#500ms;
			SC_P4_Etiketovacka.AlarmTime.PT:= T#7s;

			SC_P4_Etiketovacka.AlarmTime.IN:= NOT P4_Etiketovacka.IN.PrisavanieEtikety_Vakum_OK;

			SC_P4_Etiketovacka.IdleTime.IN:= P4_Etiketovacka.IN.PrisavanieEtikety_Vakum_OK;

			IF SC_P4_Etiketovacka.IdleTime.Q THEN
				P4_Etiketovacka.OUT.OfukEtikety_ON:= FALSE;
				SC_P4_Etiketovacka.ResetStep:= TRUE;
				SC_P4_Etiketovacka.Step:= 145;
				//			ELSIF SC_P4_Etiketovacka.AlarmTime.Q THEN
				//				P4_Etiketovacka.OUT.OfukEtikety_ON:= FALSE;
				//				P34_Alarmy[431]:= TRUE;
				//				P4_Pracovisko.STAV.Porucha_ST5:= TRUE;
			END_IF

		145:
			SC_P4_Etiketovacka.StepName:='145 - Automaticky Rezim - napolohovanie zdvihu na poziciu otocenia aplikatora';
			SC_P4_Etiketovacka.IdleTime.PT:= T#2s;
			SC_P4_Etiketovacka.AlarmTime.PT:= T#5s;

			IF NOT P4_Etiketovacka.Manual THEN
				P4_Etiketovacka.ServoZdvihuAplikatora.Parameters.Velocity:= P34_RemPremenne.P4_Etiketov_RychlZdvihuAplikat/1000;
			END_IF

			P4_Etiketovacka.ServoZdvihuAplikatora.Parameters.Position:= 255;

			IF NOT SC_P4_Etiketovacka.Switch1 AND P4_Etiketovacka.IN.Aplikator_OtocenyVZAD AND P4_Etiketovacka.IN.Aplikator_ZASUNUTY THEN
				P4_Etiketovacka.ServoZdvihuAplikatora.Command.MovePosition:= TRUE;
				SC_P4_Etiketovacka.Switch1:= TRUE;
			END_IF

			IF P4_Etiketovacka.ServoZdvihuAplikatora.Status.InPosition AND (ServoZdvihu_AktualPosition_UDINT = 255) THEN
				P4_Etiketovacka.ServoZdvihuAplikatora.Command.MovePosition:= FALSE;
				SC_P4_Etiketovacka.ResetStep:= TRUE;
				SC_P4_Etiketovacka.Step:= 148;
			END_IF

		148:
			SC_P4_Etiketovacka.StepName:='148 - Automaticky Rezim - otocenie aplikatora vpred';
			SC_P4_Etiketovacka.IdleTime.PT:= T#2s;
			SC_P4_Etiketovacka.AlarmTime.PT:= T#5s;

			IF NOT SC_P4_Etiketovacka.Switch1 THEN
				OtocAplikator_VPRED:= TRUE;
				SC_P4_Etiketovacka.Switch1:= TRUE;
			END_IF

			IF P4_Etiketovacka.IN.Aplikator_OtocenyVPRED THEN
				SC_P4_Etiketovacka.ResetStep:= TRUE;
				SC_P4_Etiketovacka.Step:= 155;
			END_IF

		155:
			SC_P4_Etiketovacka.StepName:='155 - Automaticky Rezim - napolohovanie zdvihu na poziciu nalepenia etikety';
			SC_P4_Etiketovacka.IdleTime.PT:= T#2s;
			SC_P4_Etiketovacka.AlarmTime.PT:= T#5s;

			IF NOT P4_Etiketovacka.Manual THEN
				P4_Etiketovacka.ServoZdvihuAplikatora.Parameters.Velocity:= P34_RemPremenne.P4_Etiketov_RychlZdvihuAplikat/1000;
			END_IF

			IF Linka.PAR.ZvolenyModel = '4F' THEN
				P4_Etiketovacka.ServoZdvihuAplikatora.Parameters.Position:= P34_RemPremenne.P4_Etiketovacka_PozEtikety_4F;
				ServoZdvihu_ZadanaPozicia_UDINT:= REAL_TO_UDINT(P34_RemPremenne.P4_Etiketovacka_PozEtikety_4F);
			ELSIF Linka.PAR.ZvolenyModel = '5F' THEN
				P4_Etiketovacka.ServoZdvihuAplikatora.Parameters.Position:= P34_RemPremenne.P4_Etiketovacka_PozEtikety_5F;
				ServoZdvihu_ZadanaPozicia_UDINT:= REAL_TO_UDINT(P34_RemPremenne.P4_Etiketovacka_PozEtikety_5F);
			ELSIF Linka.PAR.ZvolenyModel = '5H' THEN
				P4_Etiketovacka.ServoZdvihuAplikatora.Parameters.Position:= P34_RemPremenne.P4_Etiketovacka_PozEtikety_5H;
				ServoZdvihu_ZadanaPozicia_UDINT:= REAL_TO_UDINT(P34_RemPremenne.P4_Etiketovacka_PozEtikety_5H);
			END_IF

			IF NOT SC_P4_Etiketovacka.Switch1 AND P4_Etiketovacka.IN.Aplikator_OtocenyVPRED AND P4_Etiketovacka.IN.Aplikator_ZASUNUTY THEN
				P4_Etiketovacka.ServoZdvihuAplikatora.Command.MovePosition:= TRUE;
				SC_P4_Etiketovacka.Switch1:= TRUE;
			END_IF

			IF EDGEPOS(P4_Etiketovacka.ServoZdvihuAplikatora.Status.InPosition) THEN
				P4_Etiketovacka.ServoZdvihuAplikatora.Command.MovePosition:= FALSE;
				SC_P4_Etiketovacka.ResetStep:= TRUE;
				SC_P4_Etiketovacka.Step:= 160;
			END_IF

		160:
			SC_P4_Etiketovacka.StepName:='160 - Automaticky Rezim - vysunutie aplikatora vpred k Power CP';
			SC_P4_Etiketovacka.IdleTime.PT:= T#2s;
			SC_P4_Etiketovacka.AlarmTime.PT:= T#5s;

			IF NOT SC_P4_Etiketovacka.Switch1 THEN
				P4_Etiketovacka.OUT.Aplikator_VYSUN:= TRUE;
				SC_P4_Etiketovacka.IdleTime.IN:= TRUE;
				SC_P4_Etiketovacka.Switch1:= TRUE;
			END_IF

			IF P4_Etiketovacka.IN.Aplikator_VYSUNUTY OR SC_P4_Etiketovacka.IdleTime.Q THEN
				P4_Etiketovacka.STAV.VyrobaZacala:= TRUE;
				Paletka[i].STAV.NalepenieEtikety_DONE:= TRUE;
				SC_P4_Etiketovacka.ResetStep:= TRUE;
				SC_P4_Etiketovacka.Step:= 162;
			END_IF

		162:
			SC_P4_Etiketovacka.StepName:='162 - Automaticky Rezim - vypnutie prisavania a zasunutie aplikatora etikety';
			SC_P4_Etiketovacka.IdleTime.PT:= T#500ms;
			SC_P4_Etiketovacka.AlarmTime.PT:= T#5s;

			SC_P4_Etiketovacka.IdleTime.IN:= TRUE;

			IF NOT SC_P4_Etiketovacka.Switch1 AND SC_P4_Etiketovacka.IdleTime.Q THEN
				P4_Etiketovacka.OUT.PrisavanieEtikety_ON:= FALSE;
				P4_Etiketovacka.OUT.PrisavanieEtikety_OFF:= TRUE;
				P4_Etiketovacka.OUT.Aplikator_VYSUN:= FALSE;
				SC_P4_Etiketovacka.Switch1:= TRUE;
			END_IF

			IF P4_Etiketovacka.IN.Aplikator_ZASUNUTY THEN
				SC_P4_Etiketovacka.ResetStep:= TRUE;
				SC_P4_Etiketovacka.Step:= 168;
			END_IF

		168:
			SC_P4_Etiketovacka.StepName:='168 - Automaticky Rezim - napolohovanie zdvihu na poziciu 10mm nad etiketu';
			SC_P4_Etiketovacka.IdleTime.PT:= T#2s;
			SC_P4_Etiketovacka.AlarmTime.PT:= T#5s;

			IF NOT P4_Etiketovacka.Manual THEN
				P4_Etiketovacka.ServoZdvihuAplikatora.Parameters.Velocity:= P34_RemPremenne.P4_Etiketov_RychlZdvihuAplikat/1000;
			END_IF

			P4_Etiketovacka.ServoZdvihuAplikatora.Parameters.Position:= P4_Etiketovacka.ServoZdvihuAplikatora.Status.ActPosition - 10;

			IF NOT SC_P4_Etiketovacka.Switch1 AND P4_Etiketovacka.IN.Aplikator_ZASUNUTY THEN
				P4_Etiketovacka.ServoZdvihuAplikatora.Command.MovePosition:= TRUE;
				SC_P4_Etiketovacka.Switch1:= TRUE;
			END_IF

			IF EDGEPOS(P4_Etiketovacka.ServoZdvihuAplikatora.Status.InPosition) THEN
				P4_Etiketovacka.ServoZdvihuAplikatora.Command.MovePosition:= FALSE;
				SC_P4_Etiketovacka.ResetStep:= TRUE;
				SC_P4_Etiketovacka.Step:= 170;
			END_IF

		170:
			SC_P4_Etiketovacka.StepName:='170 - Automaticky Rezim - vysunutie aplikatora vpred k Power CP';
			SC_P4_Etiketovacka.IdleTime.PT:= T#2s;
			SC_P4_Etiketovacka.AlarmTime.PT:= T#5s;

			IF NOT SC_P4_Etiketovacka.Switch1 THEN
				P4_Etiketovacka.OUT.Aplikator_VYSUN:= TRUE;
				SC_P4_Etiketovacka.IdleTime.IN:= TRUE;
				SC_P4_Etiketovacka.Switch1:= TRUE;
			END_IF

			IF P4_Etiketovacka.IN.Aplikator_VYSUNUTY OR SC_P4_Etiketovacka.IdleTime.Q THEN
				SC_P4_Etiketovacka.ResetStep:= TRUE;
				SC_P4_Etiketovacka.Step:= 173;
			END_IF

		173:
			SC_P4_Etiketovacka.StepName:='173 - Automaticky Rezim - zasunutie aplikatora etikety';
			SC_P4_Etiketovacka.IdleTime.PT:= T#500ms;
			SC_P4_Etiketovacka.AlarmTime.PT:= T#5s;

			SC_P4_Etiketovacka.IdleTime.IN:= TRUE;

			IF NOT SC_P4_Etiketovacka.Switch1 AND SC_P4_Etiketovacka.IdleTime.Q THEN
				P4_Etiketovacka.OUT.Aplikator_VYSUN:= FALSE;
				SC_P4_Etiketovacka.Switch1:= TRUE;
			END_IF

			IF P4_Etiketovacka.IN.Aplikator_ZASUNUTY THEN
				SC_P4_Etiketovacka.ResetStep:= TRUE;
				SC_P4_Etiketovacka.Step:= 175;
			END_IF

		175:
			SC_P4_Etiketovacka.StepName:='175 - Automaticky Rezim - napolohovanie zdvihu na poziciu otocenia aplikatora';
			SC_P4_Etiketovacka.IdleTime.PT:= T#2s;
			SC_P4_Etiketovacka.AlarmTime.PT:= T#5s;

			IF NOT P4_Etiketovacka.Manual THEN
				P4_Etiketovacka.ServoZdvihuAplikatora.Parameters.Velocity:= P34_RemPremenne.P4_Etiketov_RychlZdvihuAplikat/1000;
			END_IF

			P4_Etiketovacka.ServoZdvihuAplikatora.Parameters.Position:= 255;

			IF NOT SC_P4_Etiketovacka.Switch1 THEN
				P4_Etiketovacka.ServoZdvihuAplikatora.Command.MovePosition:= TRUE;
				SC_P4_Etiketovacka.Switch1:= TRUE;
			END_IF

			IF EDGEPOS(P4_Etiketovacka.ServoZdvihuAplikatora.Status.InPosition) THEN
				P4_Etiketovacka.ServoZdvihuAplikatora.Command.MovePosition:= FALSE;
				SC_P4_Etiketovacka.ResetStep:= TRUE;
				SC_P4_Etiketovacka.Step:= 178;
			END_IF

		178:
			SC_P4_Etiketovacka.StepName:='178 - Automaticky Rezim - otocenie aplikatora vzad';
			SC_P4_Etiketovacka.IdleTime.PT:= T#2s;
			SC_P4_Etiketovacka.AlarmTime.PT:= T#5s;

			IF NOT SC_P4_Etiketovacka.Switch1 THEN
				OtocAplikator_VZAD:= TRUE;
				SC_P4_Etiketovacka.Switch1:= TRUE;
			END_IF

			IF P4_Etiketovacka.IN.Aplikator_OtocenyVZAD THEN
				SC_P4_Etiketovacka.ResetStep:= TRUE;
				SC_P4_Etiketovacka.Step:= 180;
			END_IF

		180:
			SC_P4_Etiketovacka.StepName:='180 - Automaticky Rezim - napolohovanie zdvihu na poziciu odoberania etikety';
			SC_P4_Etiketovacka.IdleTime.PT:= T#2s;
			SC_P4_Etiketovacka.AlarmTime.PT:= T#5s;

			IF NOT P4_Etiketovacka.Manual THEN
				P4_Etiketovacka.ServoZdvihuAplikatora.Parameters.Velocity:= P34_RemPremenne.P4_Etiketov_RychlZdvihuAplikat/1000;
			END_IF

			P4_Etiketovacka.ServoZdvihuAplikatora.Parameters.Position:= P34_RemPremenne.P4_Etiketovacka_PozOdoberEtikety;

			IF NOT SC_P4_Etiketovacka.Switch1 THEN
				P4_Etiketovacka.ServoZdvihuAplikatora.Command.MovePosition:= TRUE;
				SC_P4_Etiketovacka.Switch1:= TRUE;
			END_IF

			IF P4_Etiketovacka.ServoZdvihuAplikatora.Status.InPosition THEN
				P4_Etiketovacka.ServoZdvihuAplikatora.Command.MovePosition:= FALSE;
				CAM15.STAV.Results_READY:= FALSE;
				CAM15.STAV.OldRunCounter:= CAM15.STAV.RunCounter;
				IF P4_Etiketovacka.STAV.RR_SekvenciaEtiketovania_BUSY THEN
					SC_P4_Etiketovacka.ResetStep:= TRUE;
					SC_P4_Etiketovacka.Step:= 545;
				ELSE
					SC_P4_Etiketovacka.ResetStep:= TRUE;
					SC_P4_Etiketovacka.Step:= 190;
				END_IF
			END_IF

		190:
			SC_P4_Etiketovacka.StepName:='190 - Automaticky Rezim - kamerova kontrola nalepenej etikety CAM15';//CAM 15//
			SC_P4_Etiketovacka.IdleTime.PT:= T#5s;
			SC_P4_Etiketovacka.AlarmTime.PT:= T#5s;

			IF NOT SC_P4_Etiketovacka.Switch1 AND CAM15.STAV.Command_READY THEN
				CAM15.CMD.Triger:= TRUE;
				P4_Etiketovacka.STAV.Etiketa_ZhodaQRkodu_OK:= FALSE;
				SC_P4_Etiketovacka.IdleTime.IN:= TRUE;
				SC_P4_Etiketovacka.Switch1:= TRUE;
			END_IF

			IF CAM15.STAV.Results_READY AND CAM15.STAV.Command_AKCEPTOVANY AND CAM15.STAV.OldRunCounter <> CAM15.STAV.RunCounter THEN
				PocetTrigrovKamery:= 0;
				CAM15.STAV.Results_READY:= FALSE;
				CAM15.STAV.OldRunCounter:= CAM15.STAV.RunCounter;
				SC_P4_Etiketovacka.ResetStep:= TRUE;
				SC_P4_Etiketovacka.Step:= 193;
			ELSIF SC_P4_Etiketovacka.IdleTime.Q AND PocetTrigrovKamery < 5 THEN
				PocetTrigrovKamery:= PocetTrigrovKamery + 1;
				CAM15.CMD.Triger:= FALSE;
				CAM15.STAV.Results_READY:= FALSE;
				CAM15.STAV.OldRunCounter:= CAM15.STAV.RunCounter;
				SC_P4_Etiketovacka.ResetStep:= TRUE;
				SC_P4_Etiketovacka.Step:= 192;
			ELSIF SC_P4_Etiketovacka.IdleTime.Q AND PocetTrigrovKamery >= 5 THEN
				P34_Alarmy[454]:= TRUE;
				P4_Pracovisko.STAV.Porucha_ST5:= TRUE;
			END_IF

		192:
			SC_P4_Etiketovacka.StepName:='192 - Automaticky Rezim - cakam na opatovny triger kamery CAM15';
			SC_P4_Etiketovacka.IdleTime.PT:= T#1s;
			SC_P4_Etiketovacka.AlarmTime.PT:= T#5s;

			SC_P4_Etiketovacka.IdleTime.IN:= TRUE;

			IF SC_P4_Etiketovacka.IdleTime.Q THEN
				SC_P4_Etiketovacka.ResetStep:= TRUE;
				SC_P4_Etiketovacka.Step:= 190;
			END_IF

		193:
			SC_P4_Etiketovacka.StepName:='193 - Automaticky Rezim - kontrola vysledku kamery';
			SC_P4_Etiketovacka.IdleTime.PT:= T#200ms;
			SC_P4_Etiketovacka.AlarmTime.PT:= T#5s;
			SC_P4_Etiketovacka.IdleTime.IN:= TRUE;

			IF NOT CAM15.STAV.BUSY  THEN
				CAM15.CMD.Triger:= FALSE;
				IF CAM15.RESULT.CitanieQRkodu_Etikety_OK AND
					CAM15.RESULT.Pritomn_LogoBMV AND
					CAM15.RESULT.Pritomn_LogoPanasonic THEN
					SC_P4_Etiketovacka.ResetStep:= TRUE;
					SC_P4_Etiketovacka.Step:= 194;
				ELSE
					CAM15.PAR.ResultFotky:= 'FAIL';
					SC_P4_Etiketovacka.ResetStep:= TRUE;
					SC_P4_Etiketovacka.Step:= 198;
				END_IF
			END_IF

		194:
			SC_P4_Etiketovacka.StepName:='194 - Automaticky Rezim - kontrola obsahu QR kodu etikety';
			SC_P4_Etiketovacka.IdleTime.PT:= T#200ms;
			SC_P4_Etiketovacka.AlarmTime.PT:= T#5s;
			SC_P4_Etiketovacka.IdleTime.IN:= TRUE;

			IF SerioveCisloEtikety = CAM15.RESULT.PrecitanyQRkod_Etikety THEN
				P4_Etiketovacka.STAV.Etiketa_ZhodaQRkodu_OK:= TRUE;
				CAM15.PAR.ResultFotky:= 'PASS';
				SC_P4_Etiketovacka.ResetStep:= TRUE;
				SC_P4_Etiketovacka.Step:= 198;
			ELSE
				CAM15.PAR.ResultFotky:= 'FAIL';
				P4_Etiketovacka.STAV.Etiketa_ZhodaQRkodu_OK:= FALSE;
				SC_P4_Etiketovacka.ResetStep:= TRUE;
				SC_P4_Etiketovacka.Step:= 198;
			END_IF

		198:
			SC_P4_Etiketovacka.StepName:='198 - Automaticky Rezim - rozhodnutie podla kamerovej kontroly paletky';
			SC_P4_Etiketovacka.IdleTime.PT:= T#200ms;
			SC_P4_Etiketovacka.AlarmTime.PT:= T#5s;

			IF CAM15.PAR.ResultFotky = 'PASS' THEN
				Paletka[i].PAR.StavPowerCP:= 'PASS';
				SC_P4_Etiketovacka.ResetStep:= TRUE;
				SC_P4_Etiketovacka.Step:= 540;
			ELSIF CAM15.PAR.ResultFotky = 'FAIL' THEN
				P34_Vizu.ZobrazHL2_ST9:= TRUE;
				IF P4_Etiketov_KAM_Result_OK THEN
					P4_Etiketov_KAM_Result_OK:= FALSE;
					Paletka[i].PAR.StavPowerCP:= 'PASS';
					CAM15.PAR.ResultFotky:= 'PASS';
					P34_Vizu.ZobrazHL2_ST9:= FALSE;
					SC_P4_Etiketovacka.ResetStep:= TRUE;
					SC_P4_Etiketovacka.Step:= 540;
				ELSIF P4_Etiketov_KAM_Result_NG THEN
					P4_Etiketov_KAM_Result_NG:= FALSE;
					Paletka[i].PAR.StavPowerCP:= 'FAIL';
					Paletka[i].STAV.StavPaletky:= 'NG';
					P34_Vizu.ZobrazHL2_ST9:= FALSE;
					SC_P4_Etiketovacka.ResetStep:= TRUE;
					SC_P4_Etiketovacka.Step:= 540;
				END_IF
			END_IF

			//******************************Odoslanie fotiek na server***************************************//

		540:
			SC_P4_Etiketovacka.StepName:='540 - Automaticky Rezim - odoslanie fotiek na server Panasonic';
			SC_P4_Etiketovacka.IdleTime.PT:= T#200ms;
			SC_P4_Etiketovacka.AlarmTime.PT:= T#5s;

			IF Linka.KOM_FTP_OFF THEN
				SC_P4_Etiketovacka.ResetStep:= TRUE;
				SC_P4_Etiketovacka.Step:= 545;
			ELSIF NOT SC_P4_Etiketovacka.Switch1 THEN
				FTP_CAM15.INPUTS.QRkodPowerCP:= Paletka[i].PAR.QRkodPowerCP;
				CisloFotky:= CisloFotky + 1;
				FTP_CAM15.INPUTS.IndexFotky:= USINT_TO_STRING(CisloFotky);
				FTP_CAM15.INPUTS.Result:= CAM15.PAR.ResultFotky;
				Reports.Kamery.P4_CAM15_KontrolaPaletky:= CAM15.PAR.ResultFotky;
				FTP_CAM15.CMD.OdosliFotku:= TRUE;
				P4_Etiketovanie_Taktime.IN.START_MeraniaStratovehoCasu:= TRUE;
				SC_P4_Etiketovacka.Switch1:= TRUE;
			END_IF

			IF FTP_CAM15.STATUS.KomunikaciaUkoncena THEN
				FTP_CAM15.CMD.OdosliFotku:= FALSE;
				Paletka[i].STAV.OdoslanieFotiek_DONE:= TRUE;
				P4_Etiketovanie_Taktime.IN.START_MeraniaStratovehoCasu:= FALSE;
				SC_P4_Etiketovacka.ResetStep:= TRUE;
				SC_P4_Etiketovacka.Step:= 545;
			ELSIF FTP_CAM15.STATUS.KomunikaciaError THEN
				P34_Alarmy[407]:= TRUE;
				P4_Pracovisko.STAV.Porucha_ST5:= TRUE;
			END_IF

			//*************************Odcentrovanie paletky*********************************************//
		545:
			SC_P4_Etiketovacka.StepName:='545 - Automaticky Rezim - odcentrovanie paletky';
			SC_P4_Etiketovacka.IdleTime.PT:= T#200ms;
			SC_P4_Etiketovacka.AlarmTime.PT:= T#5s;

			IF NOT SC_P4_Etiketovacka.Switch1 THEN
				P4_Etiketovacka.OUT.PritlakPowerCP_VYSUN:= FALSE;
				Centrovacku_ZASUN:= TRUE;
				SC_P4_Etiketovacka.Switch1:= TRUE;
			END_IF

			IF P4_Etiketovacka.IN.Centrovanie_ZASUNUTE THEN
				IF P4_Etiketovacka.STAV.RR_SekvenciaEtiketovania_BUSY THEN
					P4_Etiketovacka.STAV.RR_SekvenciaEtiketovania_BUSY:= FALSE;
					SC_P4_Etiketovacka.ResetStep:= TRUE;
					SC_P4_Etiketovacka.Step:= 700;
				ELSE
					SC_P4_Etiketovacka.ResetStep:= TRUE;
					SC_P4_Etiketovacka.Step:= 550;
				END_IF
			END_IF

			//*******************************Odoslanie dát na server*******************************//

		550:
			SC_P4_Etiketovacka.StepName:='550 - Automaticky Rezim - odoslanie dat na server';
			SC_P4_Etiketovacka.IdleTime.PT:= T#200ms;
			SC_P4_Etiketovacka.AlarmTime.PT:= T#5s;

			IF Linka.KOM_Panatrace_OFF THEN
				SC_P4_Etiketovacka.ResetStep:= TRUE;
				SC_P4_Etiketovacka.Step:= 560;
			ELSIF NOT SC_P4_Etiketovacka.Switch1 AND TRCB_P4_Etiketovacka_ST9.STATUS.KOM_READY THEN
				TRCB_P4_Etiketovacka_ST9.CMD.OdosliStavPaletky_TYP2:= TRUE;
				(*P4_Etiketovanie_Taktime.IN.START_MeraniaStratovehoCasu:= TRUE;*)
				SC_P4_Etiketovacka.Switch1:= TRUE;
			END_IF

			IF TRCB_P4_Etiketovacka_ST9.STATUS.KomunikaciaUkoncena THEN
				TRCB_P4_Etiketovacka_ST9.CMD.OdosliStavPaletky_TYP2:= FALSE;
				P4_Etiketovanie_Taktime.IN.START_MeraniaStratovehoCasu:= FALSE;
				SC_P4_Etiketovacka.ResetStep:= TRUE;
				SC_P4_Etiketovacka.Step:= 552;
			ELSIF TRCB_P4_Etiketovacka_ST9.STATUS.KomunikaciaError THEN
				TRCB_P4_Etiketovacka_ST9.CMD.OdosliStavPaletky_TYP2:= FALSE;
				P4_Etiketovanie_Taktime.IN.START_MeraniaStratovehoCasu:= FALSE;
				SC_P4_Etiketovacka.ResetStep:= TRUE;
				SC_P4_Etiketovacka.Step:= 557;
			END_IF

		552:
			SC_P4_Etiketovacka.StepName:='552 - Automaticky Rezim - kontrola odpovede servera';
			SC_P4_Etiketovacka.IdleTime.PT:= T#200ms;
			SC_P4_Etiketovacka.AlarmTime.PT:= T#5s;

			IF NOT TRCB_P4_Etiketovacka_ST9.STATUS.KomunikaciaUkoncena THEN
				IF TRCB_P4_Etiketovacka_ST9.OUTPUTS.PovolenieCinnostiNaPaletke = 'OK' THEN
					Paletka[i].STAV.Komunikacia_DONE:= TRUE;
					P4_Etiketovacka.STAV.VyrobaZacala:= FALSE;
					SC_P4_Etiketovacka.ResetStep:= TRUE;
					SC_P4_Etiketovacka.Step:= 560;
				ELSIF TRCB_P4_Etiketovacka_ST9.OUTPUTS.PovolenieCinnostiNaPaletke = 'NG' THEN
					Paletka[i].STAV.StavPaletky:= 'NG';
					P4_Etiketovacka.STAV.VyrobaZacala:= FALSE;
					SC_P4_Etiketovacka.ResetStep:= TRUE;
					SC_P4_Etiketovacka.Step:= 560;
				END_IF
			END_IF

		555:
			SC_P4_Etiketovacka.StepName:='555 - Automaticky Rezim - vyziadanie stavu komunikacie zo serverom';
			SC_P4_Etiketovacka.IdleTime.PT:= T#200ms;
			SC_P4_Etiketovacka.AlarmTime.PT:= T#10s;

			IF NOT SC_P4_Etiketovacka.Switch1 AND TRCB_P4_Etiketovacka_ST9.STATUS.KOM_READY THEN
				TRCB_P4_Etiketovacka_ST9.CMD.VyziadajStavPanatrace_TYP4:= TRUE;
				SC_P4_Etiketovacka.Switch1:= TRUE;
			END_IF

			IF TRCB_P4_Etiketovacka_ST9.STATUS.KomunikaciaUkoncena THEN
				TRCB_P4_Etiketovacka_ST9.CMD.VyziadajStavPanatrace_TYP4:= FALSE;
				SC_P4_Etiketovacka.ResetStep:= TRUE;
				SC_P4_Etiketovacka.Step:= 556;
			ELSIF TRCB_P4_Etiketovacka_ST9.STATUS.KomunikaciaError THEN
				TRCB_P4_Etiketovacka_ST9.CMD.VyziadajStavPanatrace_TYP4:= FALSE;
				SC_P4_Etiketovacka.ResetStep:= TRUE;
				SC_P4_Etiketovacka.Step:= 557;
			END_IF

		556:
			SC_P4_Etiketovacka.StepName:='556 - Automaticky Rezim - kontrola odpovede servera';
			SC_P4_Etiketovacka.IdleTime.PT:= T#200ms;
			SC_P4_Etiketovacka.AlarmTime.PT:= T#5s;

			IF NOT TRCB_P4_Etiketovacka_ST9.STATUS.KomunikaciaUkoncena THEN
				IF TRCB_P4_Etiketovacka_ST9.OUTPUTS.DruhCinnostiNaPaletke = '0;Generating' THEN
					SC_P4_Etiketovacka.ResetStep:= TRUE;
					SC_P4_Etiketovacka.Step:= 557;
				ELSIF TRCB_P4_Etiketovacka_ST9.OUTPUTS.DruhCinnostiNaPaletke = '1;Request' THEN
					SC_P4_Etiketovacka.ResetStep:= TRUE;
					SC_P4_Etiketovacka.Step:= 557;
				ELSIF TRCB_P4_Etiketovacka_ST9.OUTPUTS.DruhCinnostiNaPaletke = '2;Report' THEN
					SC_P4_Etiketovacka.ResetStep:= TRUE;
					SC_P4_Etiketovacka.Step:= 550;
				ELSIF TRCB_P4_Etiketovacka_ST9.OUTPUTS.DruhCinnostiNaPaletke = '3;Wedding' THEN
					SC_P4_Etiketovacka.ResetStep:= TRUE;
					SC_P4_Etiketovacka.Step:= 557;
				ELSIF TRCB_P4_Etiketovacka_ST9.OUTPUTS.DruhCinnostiNaPaletke = '4;Status' THEN
					SC_P4_Etiketovacka.ResetStep:= TRUE;
					SC_P4_Etiketovacka.Step:= 557;
				ELSIF TRCB_P4_Etiketovacka_ST9.OUTPUTS.DruhCinnostiNaPaletke = '5;' THEN
					SC_P4_Etiketovacka.ResetStep:= TRUE;
					SC_P4_Etiketovacka.Step:= 557;
				ELSE
					SC_P4_Etiketovacka.ResetStep:= TRUE;
					SC_P4_Etiketovacka.Step:= 557;
				END_IF
			END_IF

		557:
			SC_P4_Etiketovacka.StepName:='557 - Automaticky Rezim - rozhodnutie obsluhy po chybe komunikacie s Panatrace';
			SC_P4_Etiketovacka.IdleTime.PT:= T#200ms;
			SC_P4_Etiketovacka.AlarmTime.PT:= T#5s;

			P34_Vizu.ZobrazHL4_ST9:= TRUE;

			IF TRCB_P4_Etiketov_OpatovnyDopyt THEN
				TRCB_P4_Etiketov_OpatovnyDopyt:= FALSE;
				P34_Vizu.ZobrazHL4_ST9:= FALSE;
				SC_P4_Etiketovacka.ResetStep:= TRUE;
				SC_P4_Etiketovacka.Step:= 555;
			ELSIF TRCB_P4_Etiketov_PaletkaNG THEN
				TRCB_P4_Etiketov_PaletkaNG:= FALSE;
				P34_Vizu.ZobrazHL4_ST9:= FALSE;
				Paletka[i].STAV.StavPaletky := 'NG';
				P4_Etiketovacka.STAV.VyrobaZacala:= FALSE;
				SC_P4_Etiketovacka.ResetStep:= TRUE;
				SC_P4_Etiketovacka.Step:= 560;
			END_IF

			//***************************Vyvezenie paletky**********************************************//

		560:
			SC_P4_Etiketovacka.StepName:='560 - Automaticky Rezim - cakam na vyvezenie na stoper vytahu';
			SC_P4_Etiketovacka.IdleTime.PT:= T#200ms;
			SC_P4_Etiketovacka.AlarmTime.PT:= T#5s;

			IF P4_Etiketovacka.KoniecCyklu THEN
				SC_P4_Etiketovacka.ResetStep:= TRUE;
				SC_P4_Etiketovacka.Step:= 0;
			ELSIF P4_Pracovisko.STAV.Porucha_ST5 THEN
				SC_P4_Etiketovacka.ResetStep:= TRUE;
				SC_P4_Etiketovacka.Step:= 0;
			ELSIF NOT P4_Vytah.RFID_hlava.PritomnostPaletky AND SC_P4_Vytah.Step = 100 AND NOT P4_Vytah.IN.PrechodDopravnika AND NOT P4_Etiketovacka.STAV.PrebiehaVyvezeniePaletky  THEN
				P4_Etiketovacka.OUT.ZasunStoper:= TRUE;
				P4_Etiketovacka.STAV.PrebiehaVyvezeniePaletky:= TRUE;
				SC_P4_Etiketovacka.ResetStep:= TRUE;
				SC_P4_Etiketovacka.Step:= 561;
			END_IF

		561:
			SC_P4_Etiketovacka.StepName:='561 - Automaticky Rezim - ukoncenie vyvazania na stoper vytahu';
			SC_P4_Etiketovacka.IdleTime.PT:= T#200ms;
			SC_P4_Etiketovacka.AlarmTime.PT:= T#10s;

			SC_P4_Etiketovacka.AlarmTime.IN:= NOT P4_Vytah.RFID_hlava.PritomnostPaletky;

			IF NOT P4_Etiketovacka.RFID_hlava.PritomnostPaletky THEN
				TestovaciKus:= FALSE;
				CisloFotky:= 0;
				Paletka[i].PAR.StavPowerCP:= '';
				Paletka[i].STAV.Komunikacia_DONE:= FALSE;
				Paletka[i].STAV.OdoslanieFotiek_DONE:= FALSE;
				Reports.Kamery.P4_CAM15_KontrolaPaletky:= '';
				P4_Etiketovacka.OUT.ZasunStoper:= FALSE;
				P4_Etiketovacka.STAV.VstupnaKamerovaKontrola:= FALSE;
			END_IF

			IF P4_Vytah.RFID_hlava.PritomnostPaletky AND NOT P4_Etiketovacka.OUT.ZasunStoper AND NOT P4_Etiketovacka.RFID_hlava.PritomnostPaletky THEN
				SC_P4_Etiketovacka.ResetStep:= TRUE;
				SC_P4_Etiketovacka.Step:= 100;
			ELSIF SC_P4_Etiketovacka.AlarmTime.Q THEN
				P34_Alarmy[452]:= TRUE;
				P4_Pracovisko.STAV.Porucha_ST5:= TRUE;
			END_IF

			//*******************************************************Manuálny režim*******************************************************************************//
		700:
			SC_P4_Etiketovacka.StepName:='700 - Manualny Rezim';
			SC_P4_Etiketovacka.IdleTime.PT:= T#8s;
			SC_P4_Etiketovacka.AlarmTime.PT:= T#5s;

			//Ovládanie zdvihu etiketovania//
			P4_Etiketovacka.ServoZdvihuAplikatora.Parameters.Acc:= 1;
			P4_Etiketovacka.ServoZdvihuAplikatora.Parameters.Dcc:= 1;
			P4_Etiketovacka.ServoZdvihuAplikatora.Parameters.Velocity:= P4_Etiketovacka.PAR.ZdvihAplikatora_JoggRychlost/1000;
			P4_Etiketovacka.ServoZdvihuAplikatora.Command.TorqueLimitation:= TRUE;
			P4_Etiketovacka.ServoZdvihuAplikatora.Parameters.Torque:= 1.5;

			IF P4_Etiketovacka.CMD.RR_ZdvihAplikatora_DOLE AND NOT P4_Etiketovacka.ServoZdvihuAplikatora.Command.Stop THEN
				P4_Etiketovacka.ServoZdvihuAplikatora.Parameters.Position:= 300;
				P4_Etiketovacka.ServoZdvihuAplikatora.Command.MovePosition:= TRUE;
			ELSIF P4_Etiketovacka.CMD.RR_ZdvihAplikatora_HORE AND NOT P4_Etiketovacka.ServoZdvihuAplikatora.Command.Stop THEN
				P4_Etiketovacka.ServoZdvihuAplikatora.Parameters.Position:= P34_RemPremenne.P4_Etiketovacka_PozOdoberEtikety;
				P4_Etiketovacka.ServoZdvihuAplikatora.Command.MovePosition:= TRUE;
			ELSE
				P4_Etiketovacka.ServoZdvihuAplikatora.Command.MovePosition:= FALSE;
				P4_Etiketovacka.ServoZdvihuAplikatora.Command.Stop:= TRUE;
			END_IF

			IF P4_Etiketovacka.ServoZdvihuAplikatora.Command.Stop AND P4_Etiketovacka.ServoZdvihuAplikatora.Status.StandStill THEN
				P4_Etiketovacka.ServoZdvihuAplikatora.Command.Stop:= FALSE;
			END_IF

			//Spustenie sekvencie nalepenia etikety//
			IF P4_Etiketovacka.CMD.RR_NalepEtiketu THEN
				P4_Etiketovacka.STAV.RR_SekvenciaEtiketovania_BUSY:= TRUE;
				P4_Etiketovacka.CMD.RR_VysunCentrovanie:= FALSE;
				P4_Etiketovacka.CMD.RR_PrisavanieEtikety:= FALSE;
				SC_P4_Etiketovacka.ResetStep:= TRUE;
				SC_P4_Etiketovacka.Step:= 118;
				P4_Etiketovacka.CMD.RR_NalepEtiketu:= FALSE;
			END_IF

			//Ovládanie zdvižky//
			IF P4_Etiketovacka.CMD.RR_VysunCentrovanie THEN
				P4_Etiketovacka.OUT.Centrovanie_ZASUN:= FALSE;
				P4_Etiketovacka.OUT.Centrovanie_VYSUN:= TRUE;
			ELSE
				P4_Etiketovacka.OUT.Centrovanie_ZASUN:= TRUE;
				P4_Etiketovacka.OUT.Centrovanie_VYSUN:= FALSE;
			END_IF

			//Prisávanie etikety//
			IF P4_Etiketovacka.CMD.RR_PrisavanieEtikety THEN
				P4_Etiketovacka.OUT.PrisavanieEtikety_OFF:= FALSE;
				P4_Etiketovacka.OUT.PrisavanieEtikety_ON:= TRUE;
			ELSE
				P4_Etiketovacka.OUT.PrisavanieEtikety_OFF:= TRUE;
				P4_Etiketovacka.OUT.PrisavanieEtikety_ON:= FALSE;
			END_IF

	END_CASE

END_PROGRAM

PROGRAM _EXIT
	(* Insert code here *)

END_PROGRAM
```

#### Types.typ - Local data types
```iecst
(**************Ovládanie tlačiarne**********************)

TYPE
	Client_typ : 	STRUCT  (*TCP Client Variables*)
		sStep : UINT; (*TCP Client Step Variable*)
		TcpOpen_0 : TcpOpen; (*AsTCP.TcpOpen FUB*)
		TcpClient_0 : TcpClient; (*AsTCP.TcpClient FUB*)
		TcpRecv_0 : TcpRecv; (*AsTCP.TcpRecv FUB*)
		TcpSend_0 : TcpSend; (*AsTCP.TcpSend FUB*)
		TcpIoctl_0 : TcpIoctl; (*AsTCP.TcpIoctl FUB*)
		TcpClose_0 : TcpClose; (*AsTCP.TcpClose FUB*)
		linger_opt : tcpLINGER_typ; (*AsTCP.tcpLINGER_typ*)
		recv_timeout : UDINT; (*receive timeout*)
		TcpOpen_timeout : UDINT;
		TcpClient_timeout : UDINT;
	END_STRUCT;
	Tlaciaren_typ : 	STRUCT
		CMD : TlaciarenCommands_typ;
		STAV : TlaciarenStatus_typ;
		Data : TlaciarenData_typ;
	END_STRUCT;
	TlaciarenCommands_typ : 	STRUCT
		VytlacEtiketu : BOOL;
	END_STRUCT;
	TlaciarenStatus_typ : 	STRUCT
		PoruchaOtvoreniaKomunikacie : BOOL;
		PoruchaOdoslaniaDat : BOOL;
		PoruchaZatvoreniaKomunikacie : BOOL;
		PoruchaSpojenia_s_Tlaciarnou : BOOL;
		PoruchaPrijatiaDat : BOOL;
		PrislaSprava_s_Tlaciarne : BOOL;
		VytlacenieEtikety_OK : BOOL;
		VytlacenieEtikety_ERROR : BOOL;
		ERROR_Number : USINT; (*1 - Porucha otvorenia komunukácie; 2 - Porucha spojenia s tlačiarnou; 3 - Porucha odoslania dat do tlačiarne; 4 - Porucha zatvorenia komunikácie;5 - Porucha prijatia dát z tlačiarne*)
	END_STRUCT;
	TlaciarenData_typ : 	STRUCT  (*Datatyp for global Variables*)
		Sprava_pre_Tlaciaren : STRING[4000]; (*Obsahuje posielane data pre tlačiareň v textovej podobe*)
		Odpoved_s_Tlaciarne : STRING[400]; (*Obsahuje odpoveď s tlačiarne*)
	END_STRUCT;
	EtiketaPanasonic_typ : 	STRUCT
		IdentificationNumber : STRING[7];
		ChangeIndex : STRING[3];
		ModelType : STRING[8];
		SupplierNumber : STRING[6];
		PlantCode : STRING[2];
		Country : STRING[2];
		Date : STRING[8];
		Counter : STRING[5];
		DataMetrix : STRING[31];
	END_STRUCT;
	Etiketa_typ : 	STRUCT
		LocationCode : STRING[2]; (*KK*)
		PartIdentNumber : STRING[7]; (*SSSSSSS*)
		ChangeIndex : STRING[2]; (*II*)
		ProductionYear : STRING[2]; (*JJ*)
		Manufactured : STRING[1]; (*H*)
		DayOfProduction : STRING[3]; (*TTT*)
		AssemblyLine : STRING[1]; (*M*)
		DayProductionCounter : STRING[5]; (*PPPPP*)
		SuplierNumber : STRING[6]; (*LLLLLL*)
		PlantCode : STRING[2]; (*NN*)
		DataMetrix : STRING[31]; (*Vytváram ho z kodu modelu na pracovisku etiketovania*)
		TypModelu : STRING[8];
		CountryCode : STRING[2];
		DatumVyroby : STRING[8]; (*02.03.20*)
	END_STRUCT;
END_TYPE
```

#### Variables.var - Local variables
```iecst
VAR
	SC_OvlCentrovacky : SequenceControlTyp;
	Centrovacku_VYSUN : BOOL;
	Centrovacku_ZASUN : BOOL;
	i : USINT;
	PocetDopytovNaServer : USINT := 0;
	SC_OvlOtacaniaAplikatora : SequenceControlTyp := (0);
	OtocAplikator_VPRED : BOOL := FALSE;
	OtocAplikator_VZAD : BOOL := FALSE;
	PocetTrigrovKamery : USINT := 0;
	CisloFotky : USINT := 0;
	TestovaciKus : BOOL := 0;
	SerioveCisloEtikety : STRING[31] := '';
	SC_OvlVysunutiaAplikatora : SequenceControlTyp := (0);
	VysunAplikator_VPRED : BOOL := FALSE;
	VysunAplikator_VZAD : BOOL := FALSE;
	ServoZdvihu_AktualPosition_UDINT : UDINT := 0;
	ServoZdvihu_ZadanaPozicia_UDINT : UDINT := 0;
END_VAR
(************Ovládanie Komunikácie s tlačiarňou*******************)
VAR
	Client : Client_typ;
	Tlaciaren : Tlaciaren_typ;
END_VAR
(************Etiketa pre Panasonic**************************)
VAR
	VstupnePoleUSINT : ARRAY[1..31] OF USINT;
	EtiketaPanasonic : EtiketaPanasonic_typ;
	Etiketa : Etiketa_typ := (0);
	CasEnable_1 : TON;
	CasResetServo_1 : TON;
	Triger_0 : BOOL := 0;
END_VAR
```

#### OvlCentrovacky.st
```iecst
ACTION OvlCentrovacky:

	//Volanie funkcie SequenceControl//
	SequenceControl(SC:= SC_OvlCentrovacky);

	CASE SC_OvlCentrovacky.Step OF

		0:
			SC_OvlCentrovacky.StepName:= '0 - Nulovanie';
			Centrovacku_VYSUN:= FALSE;
			Centrovacku_ZASUN:= FALSE;

			IF SC_P4_Etiketovacka.Step <> 0 THEN
				SC_OvlCentrovacky.ResetStep:= TRUE;
				SC_OvlCentrovacky.Step:= 1;
			END_IF

		1:
			SC_OvlCentrovacky.StepName:= '1 - Rozhodnutie o cinnosti';
			IF Centrovacku_VYSUN THEN
				SC_OvlCentrovacky.Step:= 10;
			ELSIF Centrovacku_ZASUN THEN
				SC_OvlCentrovacky.Step:= 20;
			END_IF

		10:
			SC_OvlCentrovacky.StepName:= '10 - Vysunutie centrovacky';
			SC_OvlCentrovacky.IdleTime.PT:= T#3s;
			SC_OvlCentrovacky.AlarmTime.PT:= T#6s;

			IF P4_Etiketovacka.Automat THEN
				SC_OvlCentrovacky.AlarmTime.IN:= TRUE;
			ELSE
				SC_OvlCentrovacky.IdleTime.IN:= TRUE;
			END_IF

			IF NOT SC_OvlCentrovacky.Switch1 THEN
				P4_Etiketovacka.OUT.Centrovanie_ZASUN:= FALSE;
                P4_Etiketovacka.OUT.Centrovanie_VYSUN:= TRUE;
				SC_OvlCentrovacky.Switch1:= TRUE;
			END_IF

			IF P4_Etiketovacka.IN.Centrovanie_VYSUNUTE OR SC_OvlCentrovacky.IdleTime.Q THEN
				SC_OvlCentrovacky.ResetStep:= TRUE;
				SC_OvlCentrovacky.Step:= 0;
			ELSIF SC_OvlCentrovacky.AlarmTime.Q THEN
				P34_Alarmy[404]:= TRUE;
				P4_Pracovisko.STAV.Porucha_ST5:= TRUE;
			END_IF

		20:
			SC_OvlCentrovacky.StepName:= '20 - Zasunutie centrovacky';
			SC_OvlCentrovacky.IdleTime.PT:= T#3s;
			SC_OvlCentrovacky.AlarmTime.PT:= T#6s;

			IF P4_Etiketovacka.Automat THEN
				SC_OvlCentrovacky.AlarmTime.IN:= TRUE;
			ELSE
				SC_OvlCentrovacky.IdleTime.IN:= TRUE;
			END_IF

			IF NOT SC_OvlCentrovacky.Switch1 THEN
				P4_Etiketovacka.OUT.Centrovanie_VYSUN:= FALSE;
                P4_Etiketovacka.OUT.Centrovanie_ZASUN:= TRUE;
				SC_OvlCentrovacky.Switch1:= TRUE;
			END_IF

			IF P4_Etiketovacka.IN.Centrovanie_ZASUNUTE OR SC_OvlCentrovacky.IdleTime.Q THEN
				SC_OvlCentrovacky.ResetStep:= TRUE;
				SC_OvlCentrovacky.Step:= 0;
			ELSIF SC_OvlCentrovacky.AlarmTime.Q THEN
				P34_Alarmy[405]:= TRUE;
				P4_Pracovisko.STAV.Porucha_ST5:= TRUE;
			END_IF

	END_CASE

END_ACTION
```

#### IOLinkKomunikacia.st
```iecst
ACTION IOLinkKomunikacia:

	//RFID snímač paletky//
	P4_Etiketovacka.RFID_hlava();

END_ACTION
```

#### COM_Tlaciaren.st
```iecst
ACTION COM_Tlaciaren:

	//Číslo chyby pri tlači etikety//
	//1 - Porucha otvorenia komunukácie//
	//2 - Porucha spojenia s tlačiarnou//
	//3 - Porucha odoslania dat do tlačiarne//
	//4 - Porucha zatvorenia komunikácie//
	//5 - Porucha prijatia dát z tlačiarne//

	CASE Client.sStep OF

		0://Čakanie na spustenie komunikácie z tlačiarňou//
			Tlaciaren.STAV.VytlacenieEtikety_OK:= FALSE;
			Tlaciaren.STAV.VytlacenieEtikety_ERROR:= FALSE;
			Tlaciaren.STAV.ERROR_Number:= 0;
			Tlaciaren.STAV.PrislaSprava_s_Tlaciarne:= FALSE;
			IF Tlaciaren.CMD.VytlacEtiketu THEN
				(*strcpy(ADR(Tlaciaren.Data.Sprava_pre_Tlaciaren),ADR(''));*)
				strcpy(ADR(Tlaciaren.Data.Odpoved_s_Tlaciarne),ADR('')); //Vynulovanie premennej typu string
				Client.sStep := 1;
			END_IF

		1: //Otvorenie ethernetovej komunikácie//
			Client.TcpOpen_0.enable := 1;
			Client.TcpOpen_0.pIfAddr := 0;  (* Which Interface to open *)
			Client.TcpOpen_0.port := 9100;  (* Port komunikácie s tlačiarňou *)
			Client.TcpOpen_0.options := 0;
			Client.TcpOpen_0;  (* Call the Function *)

			IF Client.TcpOpen_0.status = 0 THEN  (* TCP port je otvorený *)
				Client.TcpOpen_timeout := 0;
				Client.sStep := 5;
			ELSIF Client.TcpOpen_0.status = ERR_FUB_BUSY THEN  (* TCP port sa otvára *)
				Client.TcpOpen_timeout := Client.TcpOpen_timeout + 1;
				IF Client.TcpOpen_timeout > 50 THEN
					Tlaciaren.STAV.ERROR_Number:= 1;
					Tlaciaren.STAV.VytlacenieEtikety_ERROR:= TRUE;
					Client.TcpOpen_timeout := 0;
					Client.sStep := 40;
				END_IF
				(* Busy *)
			ELSE  (* Goto Error Step *)
				Client.TcpOpen_timeout := 0;
				Tlaciaren.STAV.ERROR_Number:= 1;
				Tlaciaren.STAV.VytlacenieEtikety_ERROR:= TRUE;
				Client.sStep := 100;
			END_IF

		5:
			Client.linger_opt.lLinger := 0; (* linger Time = 0 *)
			Client.linger_opt.lOnOff := 1; (* linger Option ON *)
			Client.TcpIoctl_0.enable := 1;
			Client.TcpIoctl_0.ident := Client.TcpOpen_0.ident; (* Connection Ident from AsTP.TCP_Open *)
			Client.TcpIoctl_0.ioctl := tcpSO_LINGER_SET; (* Set Linger Options *)
			Client.TcpIoctl_0.pData := ADR(Client.linger_opt);
			Client.TcpIoctl_0.datalen := SIZEOF(Client.linger_opt);
			Client.TcpIoctl_0;

			IF Client.TcpIoctl_0.status = 0 THEN  (* TcpIoctl successfull *)
				Client.sStep := 10;
			ELSIF Client.TcpIoctl_0.status = ERR_FUB_BUSY THEN  (* TcpIoctl not finished -> redo *)
				(* Busy *)
			ELSE  (* Goto Error Step *)
				Tlaciaren.STAV.VytlacenieEtikety_ERROR:= TRUE;
				Client.sStep := 100;
			END_IF

		10: //Spojenie s tlačiarňou//
			Client.TcpClient_0.enable := 1;
			Client.TcpClient_0.ident := Client.TcpOpen_0.ident;  (* Connection Ident from AsTCP.TCP_Open *)
			Client.TcpClient_0.portserv := 9100;  (* Port komunikácie s tlačiarňou *)
			Client.TcpClient_0.pServer := ADR('192.168.131.41');  (* Adresa tlačiarne *)
			Client.TcpClient_0;  (* Call the Function*)

			IF Client.TcpClient_0.status = 0 THEN  (* Open ok -> Send Data *)
				Client.TcpClient_timeout := 0;
				Client.sStep := 20;
			ELSIF Client.TcpClient_0.status = ERR_FUB_BUSY THEN  (* TcpClient not finished -> redo *)
				Client.TcpClient_timeout := Client.TcpClient_timeout + 1;
				IF Client.TcpClient_timeout > 50 THEN
					Tlaciaren.STAV.ERROR_Number:= 2;
					Tlaciaren.STAV.VytlacenieEtikety_ERROR:= TRUE;
					Client.TcpClient_timeout := 0;
					Client.sStep := 40;
				END_IF

				(* Busy *)
			ELSIF Client.TcpClient_0.status = tcpERR_INVALID THEN  (* Port error -> Close actual connection, and reopen a new one *)
				Client.TcpClient_timeout := 0;
				Client.sStep := 40;
			ELSE  (* Goto Error Step *)
				Client.TcpClient_timeout := 0;
				Tlaciaren.STAV.ERROR_Number:= 2;
				Tlaciaren.STAV.VytlacenieEtikety_ERROR:= TRUE;
				Client.sStep := 100;
			END_IF

		20: //Poslanie dát do tlačiarne//
			Client.TcpSend_0.enable := 1;
			Client.TcpSend_0.ident := Client.TcpOpen_0.ident;  (* Connection Ident from AsTCP.TCP_Open *)
			Client.TcpSend_0.pData := ADR(Tlaciaren.Data.Sprava_pre_Tlaciaren);  (* Dáta poslané do tlačiarne *)
			Client.TcpSend_0.datalen := SIZEOF(Tlaciaren.Data.Sprava_pre_Tlaciaren);  (* Lenght of data to send *)
			Client.TcpSend_0.flags := 0;
			Client.TcpSend_0;  (* Call the Function*)

			IF Client.TcpSend_0.status = 0 THEN  (* Data was sent sucessfully -> receive data *)
				Client.sStep := 40;
			ELSIF Client.TcpSend_0.status = ERR_FUB_BUSY THEN  (* TcpSend not finished -> redo *)
				(* Busy *)
			ELSIF (Client.TcpSend_0.status = tcpERR_SENTLEN) OR (Client.TcpSend_0.status = tcpERR_NOT_CONNECTED) THEN (* Connection Lost *)
				Client.sStep := 40;
			ELSE  (* Goto Error Step *)
				Tlaciaren.STAV.ERROR_Number:= 3;
				Tlaciaren.STAV.VytlacenieEtikety_ERROR:= TRUE;
				Client.sStep := 100;
			END_IF

		30: //Prijatie odpovede s tlačiarne//
			Client.TcpRecv_0.enable := 1;
			Client.TcpRecv_0.ident := Client.TcpOpen_0.ident;  (* Connection Ident from AsTCP.TCP_Open *)
			Client.TcpRecv_0.pData	:= ADR(Tlaciaren.Data.Odpoved_s_Tlaciarne);  (* Dáta poslané z tlačiarne *)
			Client.TcpRecv_0.datamax := SIZEOF(Tlaciaren.Data.Odpoved_s_Tlaciarne);  (* Lenght of data buffer *)
			Client.TcpRecv_0.flags := 0;
			Client.TcpRecv_0;  (* Call the Function*)

			IF Client.TcpRecv_0.status = 0 THEN  (* Data was received sucessfully -> Send next packet *)
				Tlaciaren.STAV.PrislaSprava_s_Tlaciarne:= TRUE;
				Client.recv_timeout := 0;
				Client.sStep := 40;
			ELSIF Client.TcpRecv_0.status = tcpERR_NO_DATA THEN  (* No data received - wait *)
				Client.recv_timeout := Client.recv_timeout + 1;
				IF Client.recv_timeout > 50 THEN
					Client.recv_timeout := 0;
					Client.sStep := 40;
				END_IF
				(* No Data received *)
			ELSIF Client.TcpRecv_0.status = ERR_FUB_BUSY THEN  (* TcpRecv not finished -> redo *)
				(* Busy *)
			ELSIF Client.TcpRecv_0.status = tcpERR_NOT_CONNECTED THEN (* Connection Lost *)
				Client.recv_timeout := 0;
				Client.sStep := 40;
			ELSE  (* Goto Error Step *)
				Tlaciaren.STAV.ERROR_Number:= 5;
				Tlaciaren.STAV.VytlacenieEtikety_ERROR:= TRUE;
				Client.recv_timeout := 0;
				Client.sStep := 100;
			END_IF

		40: //Zatvorenie ethernetovej komunikácie//
			Client.TcpClose_0.enable := 1;
			Client.TcpClose_0.ident := Client.TcpOpen_0.ident;  (* Connection Ident from AsTCP.TCP_Open *)
			Client.TcpClose_0.how := 0;
			Client.TcpClose_0;  (* Call the Function*)

			IF Client.TcpClose_0.status = 0 THEN  (* Close sucessfull -> Reopen the interface *)
				IF NOT Tlaciaren.STAV.VytlacenieEtikety_ERROR THEN
					Tlaciaren.STAV.VytlacenieEtikety_OK:= TRUE;
				END_IF
				Client.sStep := 100;
			ELSIF Client.TcpClose_0.status = ERR_FUB_BUSY THEN  (* TcpClose not finished -> redo *)
				(* Busy *)
			ELSE  (* Goto Error Step *)
				Tlaciaren.STAV.ERROR_Number:= 4;
				Tlaciaren.STAV.VytlacenieEtikety_ERROR:= TRUE;
				Client.sStep := 100;
			END_IF

		100: //Ukončenie komunikácie s tlačiarňou//
			IF NOT Tlaciaren.CMD.VytlacEtiketu THEN
				Client.sStep := 0;
			END_IF

	END_CASE

END_ACTION
```

#### OvlOtacaniaAplikatora.st
```iecst
ACTION OvlOtacaniaAplikatora:

	//Volanie funkcie SequenceControl//
	SequenceControl(SC:= SC_OvlOtacaniaAplikatora);

	CASE SC_OvlOtacaniaAplikatora.Step OF

		0:
			SC_OvlOtacaniaAplikatora.StepName:= '0 - Nulovanie';
			OtocAplikator_VPRED:= FALSE;
			OtocAplikator_VZAD:= FALSE;

			IF SC_P4_Etiketovacka.Step <> 0 THEN
				SC_OvlOtacaniaAplikatora.ResetStep:= TRUE;
				SC_OvlOtacaniaAplikatora.Step:= 1;
			END_IF

		1:
			SC_OvlOtacaniaAplikatora.StepName:= '1 - Rozhodnutie o cinnosti';
			IF OtocAplikator_VPRED THEN
				SC_OvlOtacaniaAplikatora.Step:= 10;
			ELSIF OtocAplikator_VZAD THEN
				SC_OvlOtacaniaAplikatora.Step:= 20;
			END_IF

		10:
			SC_OvlOtacaniaAplikatora.StepName:= '10 - Otocenie aplikatora vpred';
			SC_OvlOtacaniaAplikatora.IdleTime.PT:= T#3s;
			SC_OvlOtacaniaAplikatora.AlarmTime.PT:= T#6s;

			IF P4_Etiketovacka.Automat THEN
				SC_OvlOtacaniaAplikatora.AlarmTime.IN:= TRUE;
			ELSE
				SC_OvlOtacaniaAplikatora.IdleTime.IN:= TRUE;
			END_IF

			IF NOT SC_OvlOtacaniaAplikatora.Switch1 THEN
				P4_Etiketovacka.OUT.Aplikator_OtocVZAD:= FALSE;
                P4_Etiketovacka.OUT.Aplikator_OtocVPRED:= TRUE;
				SC_OvlOtacaniaAplikatora.Switch1:= TRUE;
			END_IF

			IF P4_Etiketovacka.IN.Aplikator_OtocenyVPRED OR SC_OvlOtacaniaAplikatora.IdleTime.Q THEN
				SC_OvlOtacaniaAplikatora.ResetStep:= TRUE;
				SC_OvlOtacaniaAplikatora.Step:= 0;
			ELSIF SC_OvlOtacaniaAplikatora.AlarmTime.Q THEN
				P34_Alarmy[462]:= TRUE;
				P4_Pracovisko.STAV.Porucha_ST5:= TRUE;
			END_IF

		20:
			SC_OvlOtacaniaAplikatora.StepName:= '20 - Otocenie aplikatora vzad';
			SC_OvlOtacaniaAplikatora.IdleTime.PT:= T#3s;
			SC_OvlOtacaniaAplikatora.AlarmTime.PT:= T#6s;

			IF P4_Etiketovacka.Automat THEN
				SC_OvlOtacaniaAplikatora.AlarmTime.IN:= TRUE;
			ELSE
				SC_OvlOtacaniaAplikatora.IdleTime.IN:= TRUE;
			END_IF

			IF NOT SC_OvlOtacaniaAplikatora.Switch1 THEN
				P4_Etiketovacka.OUT.Aplikator_OtocVPRED:= FALSE;
                P4_Etiketovacka.OUT.Aplikator_OtocVZAD:= TRUE;
				SC_OvlOtacaniaAplikatora.Switch1:= TRUE;
			END_IF

			IF P4_Etiketovacka.IN.Aplikator_OtocenyVZAD OR SC_OvlOtacaniaAplikatora.IdleTime.Q THEN
				SC_OvlOtacaniaAplikatora.ResetStep:= TRUE;
				SC_OvlOtacaniaAplikatora.Step:= 0;
			ELSIF SC_OvlOtacaniaAplikatora.AlarmTime.Q THEN
				P34_Alarmy[463]:= TRUE;
				P4_Pracovisko.STAV.Porucha_ST5:= TRUE;
			END_IF

	END_CASE

END_ACTION
```

#### VytvorenieEtikety.st
```iecst
ACTION VytvorenieEtikety:

	//*********************************************Vyčítanie parametrov etikety zo servera*******************************************************//

	brsstrcpy(ADR(VstupnePoleUSINT),ADR(SerioveCisloEtikety)); //Skopirovanie vstupnej spravy do pola

    //***************************Vyčítanie Location Code*******************************************//
    brsmemcpy(ADR(Etiketa.LocationCode),ADR(VstupnePoleUSINT[1]),2);

    //**************************Vyčítanie Part Ident Number****************************************//
    brsmemcpy(ADR(Etiketa.PartIdentNumber),ADR(VstupnePoleUSINT[3]),7);

    //**************************Vyčítanie Change Index*********************************************//
    brsmemcpy(ADR(Etiketa.ChangeIndex),ADR(VstupnePoleUSINT[10]),2);

    //**************************Vyčítanie Production Year*********************************************//
    brsmemcpy(ADR(Etiketa.ProductionYear),ADR(VstupnePoleUSINT[12]),2);

    //**************************Vyčítanie Manufactured*********************************************//
    brsmemcpy(ADR(Etiketa.Manufactured),ADR(VstupnePoleUSINT[14]),1);

    //**************************Vyčítanie Day of production*********************************************//
    brsmemcpy(ADR(Etiketa.DayOfProduction),ADR(VstupnePoleUSINT[15]),3);

    //**************************Vyčítanie Assembly line*********************************************//
    brsmemcpy(ADR(Etiketa.AssemblyLine),ADR(VstupnePoleUSINT[18]),1);

    //**************************Vyčítanie Day production counter*********************************************//
    brsmemcpy(ADR(Etiketa.DayProductionCounter),ADR(VstupnePoleUSINT[19]),5);

    //**************************Vyčítanie Supplier number*********************************************//
    brsmemcpy(ADR(Etiketa.SuplierNumber),ADR(VstupnePoleUSINT[24]),6);

    //**************************Vyčítanie Supplier plant code*********************************************//
    brsmemcpy(ADR(Etiketa.PlantCode),ADR(VstupnePoleUSINT[30]),2);

    //*****************************************************Namapovanie parametrov etikety************************************************//

    //Identification number//
    EtiketaPanasonic.IdentificationNumber:= Etiketa.PartIdentNumber;

    //Change Index//
    EtiketaPanasonic.ChangeIndex:= '';
    strcat(ADR(EtiketaPanasonic.ChangeIndex),ADR('-'));
    strcat(ADR(EtiketaPanasonic.ChangeIndex),ADR(Etiketa.ChangeIndex));

    //Model type//
    EtiketaPanasonic.ModelType:= 'POWER-CP';

    //Supplier number//
	EtiketaPanasonic.SupplierNumber:= Etiketa.SuplierNumber;

    //Plant Code//
    EtiketaPanasonic.PlantCode:= Etiketa.PlantCode;

	//Country//
	EtiketaPanasonic.Country:= 'SK';

	//Dátum//
	EtiketaPanasonic.Date:= Den_STR;
	strcat(ADR(EtiketaPanasonic.Date),ADR('.'));
	strcat(ADR(EtiketaPanasonic.Date),ADR(Mesiac_STR));
	strcat(ADR(EtiketaPanasonic.Date),ADR('.'));
	strcat(ADR(EtiketaPanasonic.Date),ADR(Rok_STR_2_Znaky));

	//Counter//
	EtiketaPanasonic.Counter:= Etiketa.DayProductionCounter;

	//Data metrix kod//
	EtiketaPanasonic.DataMetrix:= SerioveCisloEtikety;

	//***************************************Správa pre tlačiareň Compa II*************************************************//
	Tlaciaren.Data.Sprava_pre_Tlaciaren:= '^XA';//Začiatok správy
	strcat(ADR(Tlaciaren.Data.Sprava_pre_Tlaciaren),ADR('^FO210,150^A8R,40,25^FD'));
	strcat(ADR(Tlaciaren.Data.Sprava_pre_Tlaciaren),ADR(EtiketaPanasonic.IdentificationNumber));
    strcat(ADR(Tlaciaren.Data.Sprava_pre_Tlaciaren),ADR('^FS'));
    strcat(ADR(Tlaciaren.Data.Sprava_pre_Tlaciaren),ADR('^FO210,274^A8R,40,25^FD'));
    strcat(ADR(Tlaciaren.Data.Sprava_pre_Tlaciaren),ADR(EtiketaPanasonic.ChangeIndex));
    strcat(ADR(Tlaciaren.Data.Sprava_pre_Tlaciaren),ADR('^FS'));
	strcat(ADR(Tlaciaren.Data.Sprava_pre_Tlaciaren),ADR('^FO172,188^A8R,40,25^FD'));
	strcat(ADR(Tlaciaren.Data.Sprava_pre_Tlaciaren),ADR(EtiketaPanasonic.ModelType));
	strcat(ADR(Tlaciaren.Data.Sprava_pre_Tlaciaren),ADR('^FS'));
	strcat(ADR(Tlaciaren.Data.Sprava_pre_Tlaciaren),ADR('^FO134,168^A8R,40,25^FD'));
	strcat(ADR(Tlaciaren.Data.Sprava_pre_Tlaciaren),ADR(EtiketaPanasonic.SupplierNumber));
    strcat(ADR(Tlaciaren.Data.Sprava_pre_Tlaciaren),ADR('^FS'));
    strcat(ADR(Tlaciaren.Data.Sprava_pre_Tlaciaren),ADR('^FO134,290^A8R,40,25^FD'));
    strcat(ADR(Tlaciaren.Data.Sprava_pre_Tlaciaren),ADR(EtiketaPanasonic.PlantCode));
    strcat(ADR(Tlaciaren.Data.Sprava_pre_Tlaciaren),ADR('^FS'));
	strcat(ADR(Tlaciaren.Data.Sprava_pre_Tlaciaren),ADR('^FO96,290^A8R,40,25^FD'));
	strcat(ADR(Tlaciaren.Data.Sprava_pre_Tlaciaren),ADR(EtiketaPanasonic.Country));
	strcat(ADR(Tlaciaren.Data.Sprava_pre_Tlaciaren),ADR('^FS'));
	strcat(ADR(Tlaciaren.Data.Sprava_pre_Tlaciaren),ADR('^FO58,185^A8R,40,25^FD'));
	strcat(ADR(Tlaciaren.Data.Sprava_pre_Tlaciaren),ADR(EtiketaPanasonic.Date));
	strcat(ADR(Tlaciaren.Data.Sprava_pre_Tlaciaren),ADR('^FS'));
	strcat(ADR(Tlaciaren.Data.Sprava_pre_Tlaciaren),ADR('^FO20,236^A8R,40,25^FD'));
	strcat(ADR(Tlaciaren.Data.Sprava_pre_Tlaciaren),ADR(EtiketaPanasonic.Counter));
	strcat(ADR(Tlaciaren.Data.Sprava_pre_Tlaciaren),ADR('^FS'));
	strcat(ADR(Tlaciaren.Data.Sprava_pre_Tlaciaren),ADR('^FO30,40^BXR,5,200^FD'));
	strcat(ADR(Tlaciaren.Data.Sprava_pre_Tlaciaren),ADR(EtiketaPanasonic.DataMetrix));
	strcat(ADR(Tlaciaren.Data.Sprava_pre_Tlaciaren),ADR('^FS'));
	strcat(ADR(Tlaciaren.Data.Sprava_pre_Tlaciaren),ADR('^XZ'));//Koniec správy

END_ACTION
```

### Program Logical/Program/Pracovisko_4/P4_Vytah (IEC)
